// if all axes are finsihed, we're done
IF xFin AND yFin AND zFin THEN
	// reset local counters
	cX := 0;
	cY := 0;
	cZ := 0;
	fin := TRUE;
	RETURN;
END_IF

END_FUNCTION_BLOCK

// Device/Application/VG/FBs/VG_MOVE_TO_POS
(*
	Moves VG to certain position
	
Copyright (c) 2019 Manuel Goester, Michael Witt, Klaus Kammerer
Institute of Databases and Information Systems, Ulm University, Germany

Permission is hereby granted, free of charge, to any person obtaining a copy 
of this software and associated documentation files (the "Software"), to deal 
in the Software without restriction, including without limitation the rights 
to use, copy, modify, merge, publish, distribute, sublicense, and/or sell 
copies of the Software, and to permit persons to whom the Software is 
furnished to do so, subject to the following conditions:

The above copyright notice and this permission notice shall be included in 
all copies or substantial portions of the Software.

THE SOFTWARE IS PROVIDED "AS IS", WITHOUT WARRANTY OF ANY KIND, EXPRESS OR 
IMPLIED, INCLUDING BUT NOT LIMITED TO THE WARRANTIES OF MERCHANTABILITY, 
FITNESS FOR A PARTICULAR PURPOSE AND NONINFRINGEMENT. IN NO EVENT SHALL THE 
AUTHORS OR COPYRIGHT HOLDERS BE LIABLE FOR ANY CLAIM, DAMAGES OR OTHER 
LIABILITY, WHETHER IN AN ACTION OF CONTRACT, TORT OR OTHERWISE, ARISING FROM, 
OUT OF OR IN CONNECTION WITH THE SOFTWARE OR THE USE OR OTHER DEALINGS 
IN THE SOFTWARE.
*)
FUNCTION_BLOCK VG_MOVE_TO_POS
VAR_INPUT
	x: INT;
	y: INT;
	z: INT;
END_VAR
VAR_OUTPUT
END_VAR
VAR
	// finish flags
	xFin: BOOL := FALSE;
	yFin: BOOL := FALSE;
	zFin: BOOL := FALSE;
	fin: BOOL := FALSE;
	// true, if an impulse coming from the motor has been already counted
	xAlreadyCounted: BOOL := FALSE;
	yAlreadyCounted: BOOL := FALSE;
	zAlreadyCounted: BOOL := FALSE;
END_VAR

fin := FALSE;
// to handle negative counter values
IF VG.cX < 0 THEN
	VG.cX := 0;
END_IF
IF VG.cY < 0 THEN
	VG.cY := 0;
END_IF
IF VG.cZ < 0 THEN
	VG.cZ := 0;
END_IF

// X AXIS (Forward/Backward)
IF VG.cX = x THEN
	// if counter reached demanded position, we're done
	VG.mHorizontalForward := FALSE;
	VG.mHorizontalBackward := FALSE;
	xFin := TRUE;
ELSE
	xFin := FALSE;
	IF VG.cX < x AND NOT(xFin) THEN
		VG.mHorizontalForward := TRUE;
		VG.mHorizontalBackward := FALSE;
		IF VG.encHorizontal AND NOT(xAlreadyCounted) THEN
			VG.cX := VG.cX + 1;
			xAlreadyCounted := TRUE;
		ELSIF NOT(VG.encHorizontal) THEN
			xAlreadyCounted := FALSE;
		END_IF
	ELSIF VG.cX > x AND NOT(xFin) THEN
		VG.mHorizontalForward := FALSE;
		VG.mHorizontalBackward := TRUE;
		IF VG.encHorizontal AND NOT(xAlreadyCounted) THEN
			VG.cX := VG.cX - 1;
			xAlreadyCounted := TRUE;
		ELSIF NOT(VG.encHorizontal) THEN
			xAlreadyCounted := FALSE;
		END_IF
	END_IF
END_IF

// Y AXIS (Up/Down)
IF VG.cY = y THEN
	// if counter reached demanded position, we're done
	VG.mVerticalUp := FALSE;
	VG.mVerticalDown := FALSE;
	yFin := TRUE;
ELSE
	yFin := FALSE;
	IF VG.cY < y AND NOT(yFin) THEN
		VG.mVerticalDown := TRUE;
		VG.mVerticalUp := FALSE;
		IF VG.encVertical AND NOT(yAlreadyCounted) THEN
			VG.cY := VG.cY + 1;
			yAlreadyCounted := TRUE;
		ELSIF NOT(VG.encVertical) THEN
			yAlreadyCounted := FALSE;
		END_IF
	ELSIF VG.cY > y AND NOT(yFin) THEN
		VG.mVerticalUp := TRUE;
		VG.mVerticalDown := FALSE;
		IF VG.encVertical AND NOT(yAlreadyCounted) THEN
			VG.cY := VG.cY - 1;
			yAlreadyCounted := TRUE;
		ELSIF NOT(VG.encVertical) THEN
			yAlreadyCounted := FALSE;
		END_IF
	END_IF
END_IF

// Z AXIS (Rotation)
IF VG.cZ = z THEN
	// if counter reached demanded position, we're done
	VG.mRotationCClockwise := FALSE;
	VG.mRotationClockwise := FALSE;
	zFin := TRUE;
ELSE
	zFin := FALSE;
	IF VG.cZ < z AND NOT(zFin) THEN
		VG.mRotationCClockwise := TRUE;
		VG.mRotationClockwise := FALSE;
		IF VG.encRotation AND NOT(zAlreadyCounted) THEN
			VG.cZ := VG.cZ + 1;
			zAlreadyCounted := TRUE;
		ELSIF NOT(VG.encRotation) THEN
			zAlreadyCounted := FALSE;
		END_IF
	ELSIF VG.cZ > z AND NOT(zFin) THEN
		VG.mRotationCClockwise := FALSE;
		VG.mRotationClockwise := TRUE;
		IF VG.encRotation AND NOT(zAlreadyCounted) THEN
			VG.cZ := VG.cZ - 1;
			zAlreadyCounted := TRUE;
		ELSIF NOT(VG.encRotation) THEN
			zAlreadyCounted := FALSE;
		END_IF
	END_IF
END_IF

// if x and y axis are finsihed, we're done
IF xFin AND yFin AND zFin THEN
	fin := TRUE;
	RETURN;
END_IF

END_FUNCTION_BLOCK

// Device/Application/VG/VG_MULTI_MODE
PROGRAM VG_MULTI_MODE
VAR
	fin: BOOL;
	step: INT := 1;
	timer: TON;
	sorting_line_pos: INT := -1;
	vg_move_to_pos: VG_MOVE_TO_POS;
	vg_move: VG_MOVE;
END_VAR

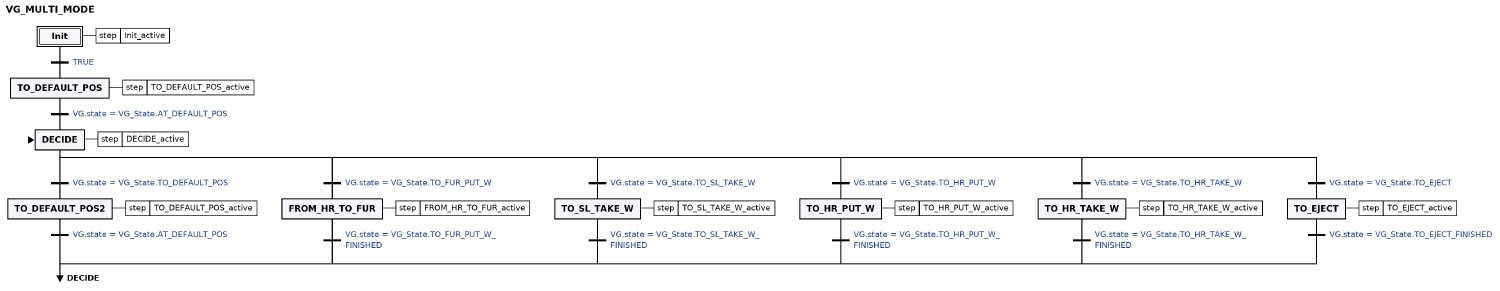
INITIAL_STEP Init:
    Init_active(N);  // step action
END_STEP
TRANSITION FROM Init TO TO_DEFAULT_POS
    := TRUE;
END_TRANSITION
STEP TO_DEFAULT_POS:
    TO_DEFAULT_POS_active(N);  // step action
END_STEP
TRANSITION FROM TO_DEFAULT_POS TO DECIDE
    := VG.state = VG_State.AT_DEFAULT_POS;
END_TRANSITION
STEP DECIDE:
    DECIDE_active(N);  // step action
END_STEP
TRANSITION FROM DECIDE TO TO_DEFAULT_POS2
    := VG.state = VG_State.TO_DEFAULT_POS;
END_TRANSITION
STEP TO_DEFAULT_POS2:
    TO_DEFAULT_POS_active(N);  // step action
END_STEP
TRANSITION FROM TO_DEFAULT_POS2 TO DECIDE
    := VG.state = VG_State.AT_DEFAULT_POS;
END_TRANSITION
TRANSITION FROM DECIDE TO FROM_HR_TO_FUR
    := VG.state = VG_State.TO_FUR_PUT_W;
END_TRANSITION
STEP FROM_HR_TO_FUR:
    FROM_HR_TO_FUR_active(N);  // step action
END_STEP
TRANSITION FROM FROM_HR_TO_FUR TO DECIDE
    := VG.state = VG_State.TO_FUR_PUT_W_FINISHED;
END_TRANSITION
TRANSITION FROM DECIDE TO TO_SL_TAKE_W
    := VG.state = VG_State.TO_SL_TAKE_W;
END_TRANSITION
STEP TO_SL_TAKE_W:
    TO_SL_TAKE_W_active(N);  // step action
END_STEP
TRANSITION FROM TO_SL_TAKE_W TO DECIDE
    := VG.state = VG_State.TO_SL_TAKE_W_FINISHED;
END_TRANSITION
TRANSITION FROM DECIDE TO TO_HR_PUT_W
    := VG.state = VG_State.TO_HR_PUT_W;
END_TRANSITION
STEP TO_HR_PUT_W:
    TO_HR_PUT_W_active(N);  // step action
END_STEP
TRANSITION FROM TO_HR_PUT_W TO DECIDE
    := VG.state = VG_State.TO_HR_PUT_W_FINISHED;
END_TRANSITION
TRANSITION FROM DECIDE TO TO_HR_TAKE_W
    := VG.state = VG_State.TO_HR_TAKE_W;
END_TRANSITION
STEP TO_HR_TAKE_W:
    TO_HR_TAKE_W_active(N);  // step action
END_STEP
TRANSITION FROM TO_HR_TAKE_W TO DECIDE
    := VG.state = VG_State.TO_HR_TAKE_W_FINISHED;
END_TRANSITION
TRANSITION FROM DECIDE TO TO_EJECT
    := VG.state = VG_State.TO_EJECT;
END_TRANSITION
STEP TO_EJECT:
    TO_EJECT_active(N);  // step action
END_STEP
TRANSITION FROM TO_EJECT TO DECIDE
    := VG.state = VG_State.TO_EJECT_FINISHED;
END_TRANSITION

ACTION TO_DEFAULT_POS_active:
(*
Copyright (c) 2019 Manuel Goester, Michael Witt, Klaus Kammerer
Institute of Databases and Information Systems, Ulm University, Germany

Permission is hereby granted, free of charge, to any person obtaining a copy 
of this software and associated documentation files (the "Software"), to deal 
in the Software without restriction, including without limitation the rights 
to use, copy, modify, merge, publish, distribute, sublicense, and/or sell 
copies of the Software, and to permit persons to whom the Software is 
furnished to do so, subject to the following conditions:

The above copyright notice and this permission notice shall be included in 
all copies or substantial portions of the Software.

THE SOFTWARE IS PROVIDED "AS IS", WITHOUT WARRANTY OF ANY KIND, EXPRESS OR 
IMPLIED, INCLUDING BUT NOT LIMITED TO THE WARRANTIES OF MERCHANTABILITY, 
FITNESS FOR A PARTICULAR PURPOSE AND NONINFRINGEMENT. IN NO EVENT SHALL THE 
AUTHORS OR COPYRIGHT HOLDERS BE LIABLE FOR ANY CLAIM, DAMAGES OR OTHER 
LIABILITY, WHETHER IN AN ACTION OF CONTRACT, TORT OR OTHERWISE, ARISING FROM, 
OUT OF OR IN CONNECTION WITH THE SOFTWARE OR THE USE OR OTHER DEALINGS 
IN THE SOFTWARE.
*)
// Brings VG to its default pos where sVertical = sHorizontal = sRotation = TRUE
// 1. y-Axis 2. z-Axis 3. rotation
IF NOT(VG.sVertical) THEN
	VG.mVerticalUp := TRUE;
ELSE
	VG.mVerticalUp := FALSE;
	// reset position counter
	VG.cY := 0;
	IF NOT(VG.sHorizontal) THEN
		VG.mHorizontalBackward := TRUE;
	ELSE
		VG.mHorizontalBackward := FALSE;
		// reset position counter
		VG.cX := 0;
		IF NOT(VG.sRotation) THEN
			VG.mRotationClockwise := TRUE;
		ELSE
			VG.mRotationClockwise := FALSE;
			// reset position counter
			VG.cZ := 0;
			
			// wait for 0.5 sec
			timer(IN:= TRUE, PT := T#0.5S);
			IF NOT(timer.Q = FALSE AND timer.IN) THEN
				timer(IN:=FALSE);
				
				// default pos reached
				VG.state := VG_State.AT_DEFAULT_POS;
			END_IF
		END_IF
	END_IF
END_IF
END_ACTION

ACTION DECIDE_active:
(*
Copyright (c) 2019 Manuel Goester, Michael Witt, Klaus Kammerer
Institute of Databases and Information Systems, Ulm University, Germany

Permission is hereby granted, free of charge, to any person obtaining a copy 
of this software and associated documentation files (the "Software"), to deal 
in the Software without restriction, including without limitation the rights 
to use, copy, modify, merge, publish, distribute, sublicense, and/or sell 
copies of the Software, and to permit persons to whom the Software is 
furnished to do so, subject to the following conditions:

The above copyright notice and this permission notice shall be included in 
all copies or substantial portions of the Software.

THE SOFTWARE IS PROVIDED "AS IS", WITHOUT WARRANTY OF ANY KIND, EXPRESS OR 
IMPLIED, INCLUDING BUT NOT LIMITED TO THE WARRANTIES OF MERCHANTABILITY, 
FITNESS FOR A PARTICULAR PURPOSE AND NONINFRINGEMENT. IN NO EVENT SHALL THE 
AUTHORS OR COPYRIGHT HOLDERS BE LIABLE FOR ANY CLAIM, DAMAGES OR OTHER 
LIABILITY, WHETHER IN AN ACTION OF CONTRACT, TORT OR OTHERWISE, ARISING FROM, 
OUT OF OR IN CONNECTION WITH THE SOFTWARE OR THE USE OR OTHER DEALINGS 
IN THE SOFTWARE.
*)
IF VG.state = VG_State.AT_HR THEN
	// this can happen if the batch job before was a single mode batch job. Then VG is already AT HR and is not in ready state
	VG.state := VG_State.TO_HR_TAKE_W;
ELSIF VG.state = VG_State.READY AND (HR.state = HR_State.GET_W AND HR.currW.state <> W_State.NULL) THEN
	// go to HR and take w
	VG.state := VG_State.TO_HR_TAKE_W;
ELSIF VG.state = VG_State.READY AND (NOT(SL.lbWhite) OR NOT(SL.lbRed) OR NOT(SL.lbBlue)) AND SL.currW.state <> W_State.NULL AND (NOT(HR.decidedToTakeANewW) OR HR.currW.state = W_State.NULL) THEN
	// go to SL and take w
	// bend VG pointers to workpiece being picked up
	VG.bIdx := SL.bIdx;
	VG.wIdx := SL.wIdx;
	VG.currW := TC.batchJobQueue.batchJobs[VG.bIdx].workpieces[VG.wIdx];
	VG.state := VG_State.TO_SL_TAKE_W;
ELSIF VG.state = VG_State.TO_SL_TAKE_W_FINISHED THEN
	// reset SL pointers
	SL.bIdx := 0;
	SL.wIdx := 0;
	SL.currW := TC.nullW;
	// at SL, w taken, decide if going to EJECT or HR
	IF VG.currW.format.ejectEnabled THEN
		// go to eject point and eject w
		VG.state := VG_State.TO_EJECT;
	ELSE
		// go to HR and put down w
		VG.state := VG_State.TO_HR_PUT_W;
	END_IF
ELSIF VG.state = VG_State.TO_HR_TAKE_W_FINISHED THEN
	// at HR, w taken, decide if going to FUR or EJECT
	IF VG.currW.format.ejectEnabled AND NOT(VG.currW.format.colorCheckEnabled OR VG.currW.format.furEnabled OR VG.currW.format.sawEnabled) THEN
		// go to eject point and eject w
		VG.state := VG_State.TO_EJECT;
	ELSE
		// go to FUR and put down w
		// but only if FUR-succer is at its default pos
		IF FUR.sSuckerPosRa THEN
			VG.state := VG_State.TO_FUR_PUT_W;
		END_IF
	END_IF
ELSIF VG.state = VG_State.TO_EJECT_FINISHED OR VG.state = VG_State.TO_FUR_PUT_W_FINISHED OR  VG.state = VG_State.TO_HR_PUT_W_FINISHED THEN
	// eject or putting w to FUR finished, back to default position for calibrating axes
	// likewise if VG put down w at HR
	VG.state := VG_State.TO_DEFAULT_POS;
ELSIF VG.state = VG_State.AT_DEFAULT_POS THEN
	// state = ready if VG is at default pos or if VG put down a w at HR --> VG is ready for next w
	VG.state := VG_state.READY;
	// reset own pointers
	VG.bIdx := 0;
	VG.wIdx := 0;
	VG.currW := TC.nullW;
END_IF
END_ACTION

ACTION FROM_HR_TO_FUR_active:
(*
Copyright (c) 2019 Manuel Goester, Michael Witt, Klaus Kammerer
Institute of Databases and Information Systems, Ulm University, Germany

Permission is hereby granted, free of charge, to any person obtaining a copy 
of this software and associated documentation files (the "Software"), to deal 
in the Software without restriction, including without limitation the rights 
to use, copy, modify, merge, publish, distribute, sublicense, and/or sell 
copies of the Software, and to permit persons to whom the Software is 
furnished to do so, subject to the following conditions:

The above copyright notice and this permission notice shall be included in 
all copies or substantial portions of the Software.

THE SOFTWARE IS PROVIDED "AS IS", WITHOUT WARRANTY OF ANY KIND, EXPRESS OR 
IMPLIED, INCLUDING BUT NOT LIMITED TO THE WARRANTIES OF MERCHANTABILITY, 
FITNESS FOR A PARTICULAR PURPOSE AND NONINFRINGEMENT. IN NO EVENT SHALL THE 
AUTHORS OR COPYRIGHT HOLDERS BE LIABLE FOR ANY CLAIM, DAMAGES OR OTHER 
LIABILITY, WHETHER IN AN ACTION OF CONTRACT, TORT OR OTHERWISE, ARISING FROM, 
OUT OF OR IN CONNECTION WITH THE SOFTWARE OR THE USE OR OTHER DEALINGS 
IN THE SOFTWARE.
*)
CASE step OF
	1:
		// x and z axis: move to FUR
		IF NOT(fin) THEN
			vg_move_to_pos(x := 131, y := 0, z := 137);
			fin := vg_move_to_pos.fin;
		ELSE
			fin := FALSE;
			step := step + 1;
		END_IF
	2:
		// y axis: move to FUR
		IF NOT(fin) THEN
			vg_move_to_pos(x := 131, y := 85, z := 137);
			fin := vg_move_to_pos.fin;
		ELSE
			fin := FALSE;
			step := step + 1;
		END_IF
	3:
		// open ventil to put down w onto waggon
		VG.valve := FALSE;
		step := step + 1;
	4:
		// wait 1 second to get sure w is not succed anymore
		timer(IN:= TRUE, PT:= T#1S);
		IF NOT(timer.Q = FALSE AND timer.IN) THEN
			// reset timer
			timer(IN:= FALSE);
			step := step + 1;
		END_IF
	5:
		// y axis: go up as far as possible
		IF NOT(VG.sVertical) THEN
			VG.mVerticalUp := TRUE;
		ELSE
			VG.mVerticalUp := FALSE;
			// reset y axis counter
			VG.cY := 0;
			// reset step counter
			step := 1;
			// bend FUR-Burner pointers to current workpiece of VG
			FUR.bIdxBurner := VG.bIdx;
			FUR.wIdxBurner := VG.wIdx;
			FUR.currWBurner := TC.batchJobQueue.batchJobs[FUR.bIdxBurner].workpieces[FUR.wIdxBurner];
			// finished
			VG.state := VG_State.TO_FUR_PUT_W_FINISHED;
		END_IF
	6:
	
END_CASE
END_ACTION

ACTION TO_SL_TAKE_W_active:
(*
Copyright (c) 2019 Manuel Goester, Michael Witt, Klaus Kammerer
Institute of Databases and Information Systems, Ulm University, Germany

Permission is hereby granted, free of charge, to any person obtaining a copy 
of this software and associated documentation files (the "Software"), to deal 
in the Software without restriction, including without limitation the rights 
to use, copy, modify, merge, publish, distribute, sublicense, and/or sell 
copies of the Software, and to permit persons to whom the Software is 
furnished to do so, subject to the following conditions:

The above copyright notice and this permission notice shall be included in 
all copies or substantial portions of the Software.

THE SOFTWARE IS PROVIDED "AS IS", WITHOUT WARRANTY OF ANY KIND, EXPRESS OR 
IMPLIED, INCLUDING BUT NOT LIMITED TO THE WARRANTIES OF MERCHANTABILITY, 
FITNESS FOR A PARTICULAR PURPOSE AND NONINFRINGEMENT. IN NO EVENT SHALL THE 
AUTHORS OR COPYRIGHT HOLDERS BE LIABLE FOR ANY CLAIM, DAMAGES OR OTHER 
LIABILITY, WHETHER IN AN ACTION OF CONTRACT, TORT OR OTHERWISE, ARISING FROM, 
OUT OF OR IN CONNECTION WITH THE SOFTWARE OR THE USE OR OTHER DEALINGS 
IN THE SOFTWARE.
*)
CASE step OF
	1:
		IF NOT(SL.currW.format.ejectEnabled) THEN
			// set flag to inform HR that VG is taking a w to bring it back to HR
			VG.storeW := TRUE;
			//VG.bIdx := SL.bIdx;
			//VG.wIdx := SL.wIdx;
			//VG.currW := TC.batchJobQueue.batchJobs[VG.bIdx].workpieces[VG.wIdx];
		END_IF
		// select sorting line pos
		IF 	TC.batchJobQueue.batchJobs[SL.bIdx].workpieces[SL.wIdx].format.colorCheckEnabled THEN
			IF TC.batchJobQueue.batchJobs[SL.bIdx].workpieces[SL.wIdx].color = 'white' AND NOT(SL.lbWhite) THEN
				sorting_line_pos := 1;
			ELSIF TC.batchJobQueue.batchJobs[SL.bIdx].workpieces[SL.wIdx].color = 'red' AND NOT(SL.lbRed) THEN
				sorting_line_pos := 2;
			ELSIF TC.batchJobQueue.batchJobs[SL.bIdx].workpieces[SL.wIdx].color = 'blue' AND NOT(SL.lbBlue) THEN
				sorting_line_pos := 3;
			END_IF
		ELSE
			// when color was not checked
			sorting_line_pos := 1;
		END_IF
		step := step + 1;
	2:
		// x and z axis: move to SL
		IF NOT(fin) THEN
			CASE sorting_line_pos OF
				1:
					vg_move_to_pos(x := 58, y := 0, z := 69);
				2:
					vg_move_to_pos(x := 63, y := 0, z := 57);
				3:
					vg_move_to_pos(x := 87, y := 0, z := 47);
			END_CASE
		fin := vg_move_to_pos.fin;
		ELSE
			fin := FALSE;
			step := step + 1;
		END_IF
	3:
		// y axis: move to SL
		IF NOT(fin) THEN
			CASE sorting_line_pos OF
				1:
					vg_move_to_pos(x := 58, y := 125, z := 69);
				2:
					vg_move_to_pos(x := 63, y := 125, z := 57);
				3:
					vg_move_to_pos(x := 87, y := 125, z := 47);
			END_CASE
		fin := vg_move_to_pos.fin;
		ELSE
			fin := FALSE;
			step := step + 1;
		END_IF
	4:
		// succ workpiece at SL
		VG.valve := TRUE;
		timer(IN:= TRUE, PT:= T#2S);
		IF timer.Q = FALSE AND timer.IN THEN
			// go
			VG.compressor := TRUE;
		ELSE
			// stop
			VG.compressor := FALSE;
			// reset timer
			timer(IN:= FALSE);
			step := step + 1;
		END_IF
	5:
		// y axis: go up as far as possible
		IF NOT(VG.sVertical) THEN
			VG.mVerticalUp := TRUE;
		ELSE
			VG.mVerticalUp := FALSE;
			// reset y axis counter
			VG.cY := 0;
			// reset step counter
			step := 1;
			// reset sorting line pos
			sorting_line_pos := -1;
			// finished
			VG.state := VG_State.TO_SL_TAKE_W_FINISHED;
		END_IF
END_CASE
END_ACTION

ACTION TO_HR_PUT_W_active:
(*
Copyright (c) 2019 Manuel Goester, Michael Witt, Klaus Kammerer
Institute of Databases and Information Systems, Ulm University, Germany

Permission is hereby granted, free of charge, to any person obtaining a copy 
of this software and associated documentation files (the "Software"), to deal 
in the Software without restriction, including without limitation the rights 
to use, copy, modify, merge, publish, distribute, sublicense, and/or sell 
copies of the Software, and to permit persons to whom the Software is 
furnished to do so, subject to the following conditions:

The above copyright notice and this permission notice shall be included in 
all copies or substantial portions of the Software.

THE SOFTWARE IS PROVIDED "AS IS", WITHOUT WARRANTY OF ANY KIND, EXPRESS OR 
IMPLIED, INCLUDING BUT NOT LIMITED TO THE WARRANTIES OF MERCHANTABILITY, 
FITNESS FOR A PARTICULAR PURPOSE AND NONINFRINGEMENT. IN NO EVENT SHALL THE 
AUTHORS OR COPYRIGHT HOLDERS BE LIABLE FOR ANY CLAIM, DAMAGES OR OTHER 
LIABILITY, WHETHER IN AN ACTION OF CONTRACT, TORT OR OTHERWISE, ARISING FROM, 
OUT OF OR IN CONNECTION WITH THE SOFTWARE OR THE USE OR OTHER DEALINGS 
IN THE SOFTWARE.
*)
CASE step OF
	1:
		// x and z axis: move to HR
		IF NOT(fin) THEN
			vg_move_to_pos(x := 27, y := 0, z := 206);
			fin := vg_move_to_pos.fin;
		ELSE
			fin := FALSE;
			step := step + 1;
		END_IF
	2:
		// box without workpiece arrived, wait 0.5 sec to be sure
		IF NOT(HR.lbOut) AND HR.state = HR_State.WAIT_FOR_VG_TO_BRING_W THEN
			timer(IN:= TRUE, PT:= T#0.5S);
			IF NOT(timer.Q = FALSE AND timer.IN) THEN
				timer(IN:= FALSE);
				step := step + 1;
			END_IF
		END_IF
	3:
		// y axis: move down at HR
		IF NOT(fin) THEN
			vg_move_to_pos(x:=27, y:=40, z:=206);
			fin := vg_move_to_pos.fin;
		ELSE
			fin := FALSE;
			step := step + 1;
		END_IF
	4:
		// open ventil
		VG.valve := FALSE;
		step := step + 1;
	5:
		timer(IN:= TRUE, PT:= T#1S);
		IF NOT(timer.Q = FALSE AND timer.IN) THEN
			// reset timer
			timer(IN:= FALSE);
			// go to next step
			step := step + 1;
		END_IF
	6:
		// y axis: go up as far as possible
		IF NOT(VG.sVertical) THEN
			VG.mVerticalUp := TRUE;
		ELSE
			VG.mVerticalUp := FALSE;
			// reset y axis counter
			VG.cY := 0;
			// reset step counter
			step := 1;
			// finished
			VG.state := VG_State.TO_HR_PUT_W_FINISHED;
		END_IF
END_CASE
END_ACTION

ACTION TO_HR_TAKE_W_active:
(*
Copyright (c) 2019 Manuel Goester, Michael Witt, Klaus Kammerer
Institute of Databases and Information Systems, Ulm University, Germany

Permission is hereby granted, free of charge, to any person obtaining a copy 
of this software and associated documentation files (the "Software"), to deal 
in the Software without restriction, including without limitation the rights 
to use, copy, modify, merge, publish, distribute, sublicense, and/or sell 
copies of the Software, and to permit persons to whom the Software is 
furnished to do so, subject to the following conditions:

The above copyright notice and this permission notice shall be included in 
all copies or substantial portions of the Software.

THE SOFTWARE IS PROVIDED "AS IS", WITHOUT WARRANTY OF ANY KIND, EXPRESS OR 
IMPLIED, INCLUDING BUT NOT LIMITED TO THE WARRANTIES OF MERCHANTABILITY, 
FITNESS FOR A PARTICULAR PURPOSE AND NONINFRINGEMENT. IN NO EVENT SHALL THE 
AUTHORS OR COPYRIGHT HOLDERS BE LIABLE FOR ANY CLAIM, DAMAGES OR OTHER 
LIABILITY, WHETHER IN AN ACTION OF CONTRACT, TORT OR OTHERWISE, ARISING FROM, 
OUT OF OR IN CONNECTION WITH THE SOFTWARE OR THE USE OR OTHER DEALINGS 
IN THE SOFTWARE.
*)
CASE step OF
	1:
		// x and z axis: move to HR
		IF NOT(fin) THEN
			vg_move_to_pos(x := 27, y := 0, z := 206);
			fin := vg_move_to_pos.fin;
		ELSE
			fin := FALSE;
			step := step + 1;
		END_IF
	2:
		IF NOT(HR.lbOut) THEN
			// box with workpiece arrived, wait 0.5 sec to be sure
			timer(IN:= TRUE, PT:= T#0.5S);
			IF NOT(timer.Q = FALSE AND timer.IN) THEN
				timer(IN:= FALSE);
				step := step + 1;
			END_IF		
		END_IF
	3:
		// y axis: move down at HR
		IF NOT(fin) THEN
			vg_move_to_pos(x:=27, y:=40, z:=206);
			fin := vg_move_to_pos.fin;
		ELSE
			fin := FALSE;
			step := step + 1;
		END_IF
	4:
		// succ w at HR
		VG.valve := TRUE;
		timer(IN:= TRUE, PT:= T#2S);
		IF timer.Q = FALSE AND timer.IN THEN
			// go
			VG.compressor := TRUE;
		ELSE
			// stop
			VG.compressor := FALSE;
			// reset timer
			timer(IN:= FALSE);
			step := step + 1;
		END_IF	
	5:
		// y axis: go up as far as possible
		IF NOT(VG.sVertical) THEN
			VG.mVerticalUp := TRUE;
		ELSE
			VG.mVerticalUp := FALSE;
			// reset y axis counter
			VG.cY := 0;
			// reset step counter
			step := 1;
			// finished
			VG.state := VG_State.TO_HR_TAKE_W_FINISHED;
		END_IF
END_CASE
END_ACTION

ACTION TO_EJECT_active:
(*
Copyright (c) 2019 Manuel Goester, Michael Witt, Klaus Kammerer
Institute of Databases and Information Systems, Ulm University, Germany

Permission is hereby granted, free of charge, to any person obtaining a copy 
of this software and associated documentation files (the "Software"), to deal 
in the Software without restriction, including without limitation the rights 
to use, copy, modify, merge, publish, distribute, sublicense, and/or sell 
copies of the Software, and to permit persons to whom the Software is 
furnished to do so, subject to the following conditions:

The above copyright notice and this permission notice shall be included in 
all copies or substantial portions of the Software.

THE SOFTWARE IS PROVIDED "AS IS", WITHOUT WARRANTY OF ANY KIND, EXPRESS OR 
IMPLIED, INCLUDING BUT NOT LIMITED TO THE WARRANTIES OF MERCHANTABILITY, 
FITNESS FOR A PARTICULAR PURPOSE AND NONINFRINGEMENT. IN NO EVENT SHALL THE 
AUTHORS OR COPYRIGHT HOLDERS BE LIABLE FOR ANY CLAIM, DAMAGES OR OTHER 
LIABILITY, WHETHER IN AN ACTION OF CONTRACT, TORT OR OTHERWISE, ARISING FROM, 
OUT OF OR IN CONNECTION WITH THE SOFTWARE OR THE USE OR OTHER DEALINGS 
IN THE SOFTWARE.
*)
CASE step OF
	1:
		// x and z axis: move to EJECT
		IF NOT(fin) THEN
			IF VG.currW.color = 'white' THEN
				// go to eject point 1
				vg_move_to_pos(x := 25, y := 0, z := 2);
			ELSIF VG.currW.color = 'red' THEN
				// go to eject point 2
				vg_move_to_pos(x := 30, y := 0, z := 15);
			ELSIF VG.currW.color = 'blue' THEN
				// go to eject point 3
				vg_move_to_pos(x := 49, y := 0, z := 23);
			ELSE
				// if color 'unknown' then eject to white eject point
				// go to eject point 1
				vg_move_to_pos(x := 25, y := 0, z := 2);
			END_IF
			fin := vg_move_to_pos.fin;
		ELSE
			fin := FALSE;
			step := step + 1;
		END_IF
	2:
		// x and z axis: move to EJECT
		IF NOT(fin) THEN
			IF VG.currW.color = 'white' THEN
				// go to eject point 1
				vg_move_to_pos(x := 25, y := 133, z := 2);
			ELSIF VG.currW.color = 'red' THEN
				// go to eject point 2
				vg_move_to_pos(x := 30, y := 133, z := 15);
			ELSIF VG.currW.color = 'blue' THEN
				// go to eject point 3
				vg_move_to_pos(x := 49, y := 133, z := 23);
			ELSE
				// if color 'unknown' then eject to white eject point
				// go to eject point 1
				vg_move_to_pos(x := 25, y := 133, z := 2);
			END_IF
			fin := vg_move_to_pos.fin;
		ELSE
			fin := FALSE;
			step := step + 1;
		END_IF
	3:
		// open valve to drop w
		VG.valve := FALSE;
		timer(IN:= TRUE, PT:= T#1S);
		IF NOT(timer.Q = FALSE AND timer.IN) THEN
			// reset timer
			timer(IN:= FALSE);
			// reset step counter
			step := 1;
			// finished
			VG.state := VG_State.TO_EJECT_FINISHED;
		END_IF
END_CASE
END_ACTION

ACTION Init_active:
(*
Copyright (c) 2019 Manuel Goester, Michael Witt, Klaus Kammerer
Institute of Databases and Information Systems, Ulm University, Germany

Permission is hereby granted, free of charge, to any person obtaining a copy 
of this software and associated documentation files (the "Software"), to deal 
in the Software without restriction, including without limitation the rights 
to use, copy, modify, merge, publish, distribute, sublicense, and/or sell 
copies of the Software, and to permit persons to whom the Software is 
furnished to do so, subject to the following conditions:

The above copyright notice and this permission notice shall be included in 
all copies or substantial portions of the Software.

THE SOFTWARE IS PROVIDED "AS IS", WITHOUT WARRANTY OF ANY KIND, EXPRESS OR 
IMPLIED, INCLUDING BUT NOT LIMITED TO THE WARRANTIES OF MERCHANTABILITY, 
FITNESS FOR A PARTICULAR PURPOSE AND NONINFRINGEMENT. IN NO EVENT SHALL THE 
AUTHORS OR COPYRIGHT HOLDERS BE LIABLE FOR ANY CLAIM, DAMAGES OR OTHER 
LIABILITY, WHETHER IN AN ACTION OF CONTRACT, TORT OR OTHERWISE, ARISING FROM, 
OUT OF OR IN CONNECTION WITH THE SOFTWARE OR THE USE OR OTHER DEALINGS 
IN THE SOFTWARE.
*)
step := 1;
END_ACTION

END_PROGRAM

// Device/Application/SL/SL_SINGLE_MODE
PROGRAM SL_SINGLE_MODE
VAR
	sl_fb: SL_FB;
	step: INT := 1;
	fin: BOOL;
END_VAR

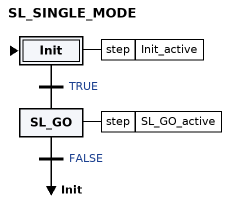
INITIAL_STEP Init:
    Init_active(N);  // step action
END_STEP
TRANSITION FROM Init TO SL_GO
    := TRUE;
END_TRANSITION
STEP SL_GO:
    SL_GO_active(N);  // step action
END_STEP
TRANSITION FROM SL_GO TO Init
    := FALSE;
END_TRANSITION

ACTION Init_active:
(*
Copyright (c) 2019 Manuel Goester, Michael Witt, Klaus Kammerer
Institute of Databases and Information Systems, Ulm University, Germany

Permission is hereby granted, free of charge, to any person obtaining a copy 
of this software and associated documentation files (the "Software"), to deal 
in the Software without restriction, including without limitation the rights 
to use, copy, modify, merge, publish, distribute, sublicense, and/or sell 
copies of the Software, and to permit persons to whom the Software is 
furnished to do so, subject to the following conditions:

The above copyright notice and this permission notice shall be included in 
all copies or substantial portions of the Software.

THE SOFTWARE IS PROVIDED "AS IS", WITHOUT WARRANTY OF ANY KIND, EXPRESS OR 
IMPLIED, INCLUDING BUT NOT LIMITED TO THE WARRANTIES OF MERCHANTABILITY, 
FITNESS FOR A PARTICULAR PURPOSE AND NONINFRINGEMENT. IN NO EVENT SHALL THE 
AUTHORS OR COPYRIGHT HOLDERS BE LIABLE FOR ANY CLAIM, DAMAGES OR OTHER 
LIABILITY, WHETHER IN AN ACTION OF CONTRACT, TORT OR OTHERWISE, ARISING FROM, 
OUT OF OR IN CONNECTION WITH THE SOFTWARE OR THE USE OR OTHER DEALINGS 
IN THE SOFTWARE.
*)
SL.state := SL_State.WAITING_FOR_W;
END_ACTION

ACTION SL_GO_active:
(*
Copyright (c) 2019 Manuel Goester, Michael Witt, Klaus Kammerer
Institute of Databases and Information Systems, Ulm University, Germany

Permission is hereby granted, free of charge, to any person obtaining a copy 
of this software and associated documentation files (the "Software"), to deal 
in the Software without restriction, including without limitation the rights 
to use, copy, modify, merge, publish, distribute, sublicense, and/or sell 
copies of the Software, and to permit persons to whom the Software is 
furnished to do so, subject to the following conditions:

The above copyright notice and this permission notice shall be included in 
all copies or substantial portions of the Software.

THE SOFTWARE IS PROVIDED "AS IS", WITHOUT WARRANTY OF ANY KIND, EXPRESS OR 
IMPLIED, INCLUDING BUT NOT LIMITED TO THE WARRANTIES OF MERCHANTABILITY, 
FITNESS FOR A PARTICULAR PURPOSE AND NONINFRINGEMENT. IN NO EVENT SHALL THE 
AUTHORS OR COPYRIGHT HOLDERS BE LIABLE FOR ANY CLAIM, DAMAGES OR OTHER 
LIABILITY, WHETHER IN AN ACTION OF CONTRACT, TORT OR OTHERWISE, ARISING FROM, 
OUT OF OR IN CONNECTION WITH THE SOFTWARE OR THE USE OR OTHER DEALINGS 
IN THE SOFTWARE.
*)
CASE step OF
	1:
		IF SL.state = SL_State.W_RECEIVED THEN
			step := step + 1;
		END_IF
	2:
		IF NOT(fin) THEN
			sl_fb();
			fin := sl_fb.fin;
		ELSE
			// wait for VG to pick up w
			SL.state := SL_State.WAITING_FOR_VG_TO_PICK_UP_W;
			step := step + 1;
		END_IF
	3:
		// reset own pointers
		SL.bIdx := 0;
		SL.wIdx := 0;
		// reset fin
		fin := FALSE;
		step := 1;
		SL.state := SL_State.WAITING_FOR_W;
END_CASE
END_ACTION

END_PROGRAM

// Device/Application/SL/FBs/SL_FB
(*
	Implements the functionality of sorting line
*)
FUNCTION_BLOCK SL_FB
VAR_INPUT
END_VAR
VAR_OUTPUT
END_VAR
VAR
	trigger : INT;
	puls_temp : INT := 0;
	counter_puls : INT;
	white : BOOL;
	red : BOOL;
	blue : BOOL;
	
	color_value : DINT;
	
	rack_white : INT := 0;
	rack_red : INT := 0;
	rack_blue : INT := 0;
	
	timer : TON;
	passed: BOOL;
	fin: BOOL;
END_VAR

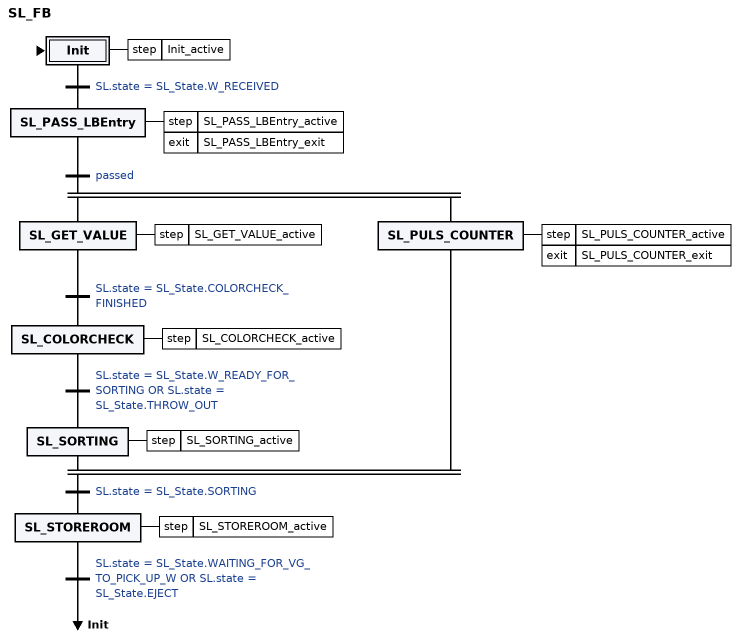
INITIAL_STEP Init:
    Init_active(N);  // step action
END_STEP
TRANSITION FROM Init TO SL_PASS_LBEntry
    := SL.state = SL_State.W_RECEIVED;
END_TRANSITION
STEP SL_PASS_LBEntry:
    SL_PASS_LBEntry_active(N);  // step action
    SL_PASS_LBEntry_exit(P0);  // exit action
END_STEP
TRANSITION FROM SL_PASS_LBEntry TO (SL_GET_VALUE, SL_PULS_COUNTER)
    := passed;
END_TRANSITION
STEP SL_GET_VALUE:
    SL_GET_VALUE_active(N);  // step action
END_STEP
TRANSITION FROM SL_GET_VALUE TO SL_COLORCHECK
    := SL.state = SL_State.COLORCHECK_FINISHED;
END_TRANSITION
STEP SL_COLORCHECK:
    SL_COLORCHECK_active(N);  // step action
END_STEP
TRANSITION FROM SL_COLORCHECK TO SL_SORTING
    := SL.state = SL_State.W_READY_FOR_SORTING OR SL.state = SL_State.THROW_OUT;
END_TRANSITION
STEP SL_SORTING:
    SL_SORTING_active(N);  // step action
END_STEP
STEP SL_PULS_COUNTER:
    SL_PULS_COUNTER_active(N);  // step action
    SL_PULS_COUNTER_exit(P0);  // exit action
END_STEP
TRANSITION FROM (SL_SORTING, SL_PULS_COUNTER) TO SL_STOREROOM
    := SL.state = SL_State.SORTING;
END_TRANSITION
STEP SL_STOREROOM:
    SL_STOREROOM_active(N);  // step action
END_STEP
TRANSITION FROM SL_STOREROOM TO Init
    := SL.state = SL_State.WAITING_FOR_VG_TO_PICK_UP_W OR SL.state = SL_State.EJECT;
END_TRANSITION

ACTION Init_active:
(*
Copyright (c) 2019 Manuel Goester, Michael Witt, Klaus Kammerer
Institute of Databases and Information Systems, Ulm University, Germany

Permission is hereby granted, free of charge, to any person obtaining a copy 
of this software and associated documentation files (the "Software"), to deal 
in the Software without restriction, including without limitation the rights 
to use, copy, modify, merge, publish, distribute, sublicense, and/or sell 
copies of the Software, and to permit persons to whom the Software is 
furnished to do so, subject to the following conditions:

The above copyright notice and this permission notice shall be included in 
all copies or substantial portions of the Software.

THE SOFTWARE IS PROVIDED "AS IS", WITHOUT WARRANTY OF ANY KIND, EXPRESS OR 
IMPLIED, INCLUDING BUT NOT LIMITED TO THE WARRANTIES OF MERCHANTABILITY, 
FITNESS FOR A PARTICULAR PURPOSE AND NONINFRINGEMENT. IN NO EVENT SHALL THE 
AUTHORS OR COPYRIGHT HOLDERS BE LIABLE FOR ANY CLAIM, DAMAGES OR OTHER 
LIABILITY, WHETHER IN AN ACTION OF CONTRACT, TORT OR OTHERWISE, ARISING FROM, 
OUT OF OR IN CONNECTION WITH THE SOFTWARE OR THE USE OR OTHER DEALINGS 
IN THE SOFTWARE.
*)
trigger := 0;
puls_temp := 0;
counter_puls := 0;
white := FALSE;
red := FALSE;
blue := FALSE;

color_value := 4000000;

timer(IN:=FALSE);
fin := FALSE;

SL.mConveyorBelt := TRUE;
END_ACTION

ACTION SL_COLORCHECK_active:
(*
Copyright (c) 2019 Manuel Goester, Michael Witt, Klaus Kammerer
Institute of Databases and Information Systems, Ulm University, Germany

Permission is hereby granted, free of charge, to any person obtaining a copy 
of this software and associated documentation files (the "Software"), to deal 
in the Software without restriction, including without limitation the rights 
to use, copy, modify, merge, publish, distribute, sublicense, and/or sell 
copies of the Software, and to permit persons to whom the Software is 
furnished to do so, subject to the following conditions:

The above copyright notice and this permission notice shall be included in 
all copies or substantial portions of the Software.

THE SOFTWARE IS PROVIDED "AS IS", WITHOUT WARRANTY OF ANY KIND, EXPRESS OR 
IMPLIED, INCLUDING BUT NOT LIMITED TO THE WARRANTIES OF MERCHANTABILITY, 
FITNESS FOR A PARTICULAR PURPOSE AND NONINFRINGEMENT. IN NO EVENT SHALL THE 
AUTHORS OR COPYRIGHT HOLDERS BE LIABLE FOR ANY CLAIM, DAMAGES OR OTHER 
LIABILITY, WHETHER IN AN ACTION OF CONTRACT, TORT OR OTHERWISE, ARISING FROM, 
OUT OF OR IN CONNECTION WITH THE SOFTWARE OR THE USE OR OTHER DEALINGS 
IN THE SOFTWARE.
*)
IF color_value > 2000000 AND color_value < 2558000 THEN//weis: 2630000
	TC.batchJobQueue.batchJobs[SL.bIdx].workpieces[SL.wIdx].color := 'white';
	white := TRUE;
	red := FALSE;
	blue := FALSE;
	SL.state := SL_State.W_READY_FOR_SORTING;
END_IF
IF color_value > 2558001 AND color_value < 3000000 THEN//rot: 2801000
	TC.batchJobQueue.batchJobs[SL.bIdx].workpieces[SL.wIdx].color := 'red';
	white := FALSE;
	red := TRUE;
	blue := FALSE;
	SL.state := SL_State.W_READY_FOR_SORTING;
END_IF
IF color_value > 3400000 AND color_value < 3600000 THEN//blau: 3546000
	TC.batchJobQueue.batchJobs[SL.bIdx].workpieces[SL.wIdx].color := 'blue';
	white := FALSE;
	red := FALSE;
	blue := TRUE;
	SL.state := SL_State.W_READY_FOR_SORTING;
END_IF
IF color_value > 3600000 OR color_value < 2000000 THEN//unknown
	TC.batchJobQueue.batchJobs[SL.bIdx].workpieces[SL.wIdx].color := 'unknown';
	white := FALSE;
	red := FALSE;
	blue := FALSE;
	SL.state := SL_State.THROW_OUT; 
END_IF

SL.mConveyorBelt := TRUE;
END_ACTION

ACTION SL_GET_VALUE_active:
(*
Copyright (c) 2019 Manuel Goester, Michael Witt, Klaus Kammerer
Institute of Databases and Information Systems, Ulm University, Germany

Permission is hereby granted, free of charge, to any person obtaining a copy 
of this software and associated documentation files (the "Software"), to deal 
in the Software without restriction, including without limitation the rights 
to use, copy, modify, merge, publish, distribute, sublicense, and/or sell 
copies of the Software, and to permit persons to whom the Software is 
furnished to do so, subject to the following conditions:

The above copyright notice and this permission notice shall be included in 
all copies or substantial portions of the Software.

THE SOFTWARE IS PROVIDED "AS IS", WITHOUT WARRANTY OF ANY KIND, EXPRESS OR 
IMPLIED, INCLUDING BUT NOT LIMITED TO THE WARRANTIES OF MERCHANTABILITY, 
FITNESS FOR A PARTICULAR PURPOSE AND NONINFRINGEMENT. IN NO EVENT SHALL THE 
AUTHORS OR COPYRIGHT HOLDERS BE LIABLE FOR ANY CLAIM, DAMAGES OR OTHER 
LIABILITY, WHETHER IN AN ACTION OF CONTRACT, TORT OR OTHERWISE, ARISING FROM, 
OUT OF OR IN CONNECTION WITH THE SOFTWARE OR THE USE OR OTHER DEALINGS 
IN THE SOFTWARE.
*)
IF NOT(SL.lbAfterColorSensor) THEN
	SL.state := SL_State.COLORCHECK_FINISHED;
ELSE
	SL.state := SL_State.W_AT_COLORCHECK;
	IF SL.colorSensor < color_value THEN
		color_value := SL.colorSensor;
	END_IF
END_IF 

SL.mConveyorBelt := TRUE;
END_ACTION

ACTION SL_PASS_LBEntry_active:
(*
Copyright (c) 2019 Manuel Goester, Michael Witt, Klaus Kammerer
Institute of Databases and Information Systems, Ulm University, Germany

Permission is hereby granted, free of charge, to any person obtaining a copy 
of this software and associated documentation files (the "Software"), to deal 
in the Software without restriction, including without limitation the rights 
to use, copy, modify, merge, publish, distribute, sublicense, and/or sell 
copies of the Software, and to permit persons to whom the Software is 
furnished to do so, subject to the following conditions:

The above copyright notice and this permission notice shall be included in 
all copies or substantial portions of the Software.

THE SOFTWARE IS PROVIDED "AS IS", WITHOUT WARRANTY OF ANY KIND, EXPRESS OR 
IMPLIED, INCLUDING BUT NOT LIMITED TO THE WARRANTIES OF MERCHANTABILITY, 
FITNESS FOR A PARTICULAR PURPOSE AND NONINFRINGEMENT. IN NO EVENT SHALL THE 
AUTHORS OR COPYRIGHT HOLDERS BE LIABLE FOR ANY CLAIM, DAMAGES OR OTHER 
LIABILITY, WHETHER IN AN ACTION OF CONTRACT, TORT OR OTHERWISE, ARISING FROM, 
OUT OF OR IN CONNECTION WITH THE SOFTWARE OR THE USE OR OTHER DEALINGS 
IN THE SOFTWARE.
*)
IF NOT(SL.lbEntry) AND trigger < 1 THEN
	trigger := trigger + 1;
	SL.state := SL_State.W_AT_LB;
END_IF

IF lbEntry AND trigger >= 1 THEN
	passed := TRUE;
END_IF

SL.mConveyorBelt := TRUE;
END_ACTION

ACTION SL_PASS_LBEntry_exit:
(*
Copyright (c) 2019 Manuel Goester, Michael Witt, Klaus Kammerer
Institute of Databases and Information Systems, Ulm University, Germany

Permission is hereby granted, free of charge, to any person obtaining a copy 
of this software and associated documentation files (the "Software"), to deal 
in the Software without restriction, including without limitation the rights 
to use, copy, modify, merge, publish, distribute, sublicense, and/or sell 
copies of the Software, and to permit persons to whom the Software is 
furnished to do so, subject to the following conditions:

The above copyright notice and this permission notice shall be included in 
all copies or substantial portions of the Software.

THE SOFTWARE IS PROVIDED "AS IS", WITHOUT WARRANTY OF ANY KIND, EXPRESS OR 
IMPLIED, INCLUDING BUT NOT LIMITED TO THE WARRANTIES OF MERCHANTABILITY, 
FITNESS FOR A PARTICULAR PURPOSE AND NONINFRINGEMENT. IN NO EVENT SHALL THE 
AUTHORS OR COPYRIGHT HOLDERS BE LIABLE FOR ANY CLAIM, DAMAGES OR OTHER 
LIABILITY, WHETHER IN AN ACTION OF CONTRACT, TORT OR OTHERWISE, ARISING FROM, 
OUT OF OR IN CONNECTION WITH THE SOFTWARE OR THE USE OR OTHER DEALINGS 
IN THE SOFTWARE.
*)
passed := FALSE;
puls_temp := 0;
counter_puls := 0;
END_ACTION

ACTION SL_PULS_COUNTER_active:
(*
Copyright (c) 2019 Manuel Goester, Michael Witt, Klaus Kammerer
Institute of Databases and Information Systems, Ulm University, Germany

Permission is hereby granted, free of charge, to any person obtaining a copy 
of this software and associated documentation files (the "Software"), to deal 
in the Software without restriction, including without limitation the rights 
to use, copy, modify, merge, publish, distribute, sublicense, and/or sell 
copies of the Software, and to permit persons to whom the Software is 
furnished to do so, subject to the following conditions:

The above copyright notice and this permission notice shall be included in 
all copies or substantial portions of the Software.

THE SOFTWARE IS PROVIDED "AS IS", WITHOUT WARRANTY OF ANY KIND, EXPRESS OR 
IMPLIED, INCLUDING BUT NOT LIMITED TO THE WARRANTIES OF MERCHANTABILITY, 
FITNESS FOR A PARTICULAR PURPOSE AND NONINFRINGEMENT. IN NO EVENT SHALL THE 
AUTHORS OR COPYRIGHT HOLDERS BE LIABLE FOR ANY CLAIM, DAMAGES OR OTHER 
LIABILITY, WHETHER IN AN ACTION OF CONTRACT, TORT OR OTHERWISE, ARISING FROM, 
OUT OF OR IN CONNECTION WITH THE SOFTWARE OR THE USE OR OTHER DEALINGS 
IN THE SOFTWARE.
*)
//count convoyorbelt buttons
IF SL.mConveyorBelt AND SL.iFeeler THEN //button push
	IF puls_temp = 0 THEN
		counter_puls := counter_puls +1;
	END_IF
	
	puls_temp := puls_temp +1;
END_IF

IF puls_temp > 0 AND SL.mConveyorBelt AND NOT(iFeeler) THEN // button release
	puls_temp := 0;
	counter_puls := counter_puls +1;
END_IF
END_ACTION

ACTION SL_PULS_COUNTER_exit:
(*
Copyright (c) 2019 Manuel Goester, Michael Witt, Klaus Kammerer
Institute of Databases and Information Systems, Ulm University, Germany

Permission is hereby granted, free of charge, to any person obtaining a copy 
of this software and associated documentation files (the "Software"), to deal 
in the Software without restriction, including without limitation the rights 
to use, copy, modify, merge, publish, distribute, sublicense, and/or sell 
copies of the Software, and to permit persons to whom the Software is 
furnished to do so, subject to the following conditions:

The above copyright notice and this permission notice shall be included in 
all copies or substantial portions of the Software.

THE SOFTWARE IS PROVIDED "AS IS", WITHOUT WARRANTY OF ANY KIND, EXPRESS OR 
IMPLIED, INCLUDING BUT NOT LIMITED TO THE WARRANTIES OF MERCHANTABILITY, 
FITNESS FOR A PARTICULAR PURPOSE AND NONINFRINGEMENT. IN NO EVENT SHALL THE 
AUTHORS OR COPYRIGHT HOLDERS BE LIABLE FOR ANY CLAIM, DAMAGES OR OTHER 
LIABILITY, WHETHER IN AN ACTION OF CONTRACT, TORT OR OTHERWISE, ARISING FROM, 
OUT OF OR IN CONNECTION WITH THE SOFTWARE OR THE USE OR OTHER DEALINGS 
IN THE SOFTWARE.
*)
counter_puls := 0;
puls_temp := 0;
END_ACTION

ACTION SL_SORTING_active:
(*
Copyright (c) 2019 Manuel Goester, Michael Witt, Klaus Kammerer
Institute of Databases and Information Systems, Ulm University, Germany

Permission is hereby granted, free of charge, to any person obtaining a copy 
of this software and associated documentation files (the "Software"), to deal 
in the Software without restriction, including without limitation the rights 
to use, copy, modify, merge, publish, distribute, sublicense, and/or sell 
copies of the Software, and to permit persons to whom the Software is 
furnished to do so, subject to the following conditions:

The above copyright notice and this permission notice shall be included in 
all copies or substantial portions of the Software.

THE SOFTWARE IS PROVIDED "AS IS", WITHOUT WARRANTY OF ANY KIND, EXPRESS OR 
IMPLIED, INCLUDING BUT NOT LIMITED TO THE WARRANTIES OF MERCHANTABILITY, 
FITNESS FOR A PARTICULAR PURPOSE AND NONINFRINGEMENT. IN NO EVENT SHALL THE 
AUTHORS OR COPYRIGHT HOLDERS BE LIABLE FOR ANY CLAIM, DAMAGES OR OTHER 
LIABILITY, WHETHER IN AN ACTION OF CONTRACT, TORT OR OTHERWISE, ARISING FROM, 
OUT OF OR IN CONNECTION WITH THE SOFTWARE OR THE USE OR OTHER DEALINGS 
IN THE SOFTWARE.
*)
SL.mConveyorBelt := TRUE;
IF TC.batchJobQueue.batchJobs[SL.bIdx].workpieces[SL.wIdx].format.colorCheckEnabled THEN
	timer(IN:= TRUE, PT := T#3S);
	IF white AND counter_puls = 35 THEN
		SL.mConveyorBelt := FALSE;
		SL.compressor := TRUE;
		SL.valveFirstEject := TRUE;
	END_IF
	
	IF red AND counter_puls = 45 THEN
		SL.mConveyorBelt := FALSE;
		SL.compressor := TRUE;
		SL.valveSecEject := TRUE;
	END_IF
	
	IF blue AND counter_puls = 55 THEN
		SL.mConveyorBelt := FALSE;
		SL.compressor := TRUE;
		SL.valveThirdEject := TRUE;
	END_IF
	
	IF NOT(timer.Q = FALSE AND timer.IN) THEN
		SL.mConveyorBelt := FALSE;
		SL.compressor := FALSE;	
		SL.valveFirstEject := FALSE;
		SL.valveSecEject := FALSE;
		SL.valveThirdEject := FALSE;
		
		timer(IN:= FALSE);
		
		SL.state := SL_State.SORTING;
	END_IF
ELSE
	timer(IN:= TRUE, PT := T#2S);
	IF counter_puls = 37 THEN
		SL.mConveyorBelt := FALSE;
		SL.compressor := TRUE;
		SL.valveFirstEject := TRUE;
	END_IF
	IF NOT(timer.Q = FALSE AND timer.IN) THEN
		SL.compressor := FALSE;	
		SL.valveFirstEject := FALSE;
		SL.valveSecEject := FALSE;
		SL.valveThirdEject := FALSE;
		
		timer(IN:= FALSE);
		
		SL.state := SL_State.SORTING;
	END_IF
END_IF
END_ACTION

ACTION SL_STOREROOM_active:
(*
Copyright (c) 2019 Manuel Goester, Michael Witt, Klaus Kammerer
Institute of Databases and Information Systems, Ulm University, Germany

Permission is hereby granted, free of charge, to any person obtaining a copy 
of this software and associated documentation files (the "Software"), to deal 
in the Software without restriction, including without limitation the rights 
to use, copy, modify, merge, publish, distribute, sublicense, and/or sell 
copies of the Software, and to permit persons to whom the Software is 
furnished to do so, subject to the following conditions:

The above copyright notice and this permission notice shall be included in 
all copies or substantial portions of the Software.

THE SOFTWARE IS PROVIDED "AS IS", WITHOUT WARRANTY OF ANY KIND, EXPRESS OR 
IMPLIED, INCLUDING BUT NOT LIMITED TO THE WARRANTIES OF MERCHANTABILITY, 
FITNESS FOR A PARTICULAR PURPOSE AND NONINFRINGEMENT. IN NO EVENT SHALL THE 
AUTHORS OR COPYRIGHT HOLDERS BE LIABLE FOR ANY CLAIM, DAMAGES OR OTHER 
LIABILITY, WHETHER IN AN ACTION OF CONTRACT, TORT OR OTHERWISE, ARISING FROM, 
OUT OF OR IN CONNECTION WITH THE SOFTWARE OR THE USE OR OTHER DEALINGS 
IN THE SOFTWARE.
*)
IF white AND NOT(SL.lbWhite) THEN
	rack_white := rack_white + 1;
	SL.state := SL_State.WAITING_FOR_VG_TO_PICK_UP_W;
ELSIF red AND NOT(SL.lbRed) THEN
	rack_red := rack_red + 1;
	SL.state := SL_State.WAITING_FOR_VG_TO_PICK_UP_W;
ELSIF blue AND NOT(SL.lbBlue) THEN
	rack_blue := rack_blue + 1;
	SL.state := SL_State.WAITING_FOR_VG_TO_PICK_UP_W;
ELSE
	// no sorting
	SL.state := SL_State.EJECT;
END_IF
// important! --> signals SL_single/multi_MODE PRG that FB is finished
fin := TRUE;
END_ACTION

END_FUNCTION_BLOCK

// Device/Application/SL/SL_MULTI_MODE
PROGRAM SL_MULTI_MODE
VAR
	fin: BOOL;
	sl_fb: SL_FB;
	step: INT := 1;
END_VAR

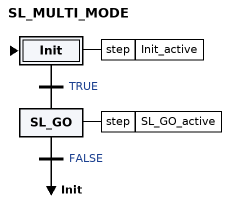
INITIAL_STEP Init:
    Init_active(N);  // step action
END_STEP
TRANSITION FROM Init TO SL_GO
    := TRUE;
END_TRANSITION
STEP SL_GO:
    SL_GO_active(N);  // step action
END_STEP
TRANSITION FROM SL_GO TO Init
    := FALSE;
END_TRANSITION

ACTION SL_GO_active:
(*
Copyright (c) 2019 Manuel Goester, Michael Witt, Klaus Kammerer
Institute of Databases and Information Systems, Ulm University, Germany

Permission is hereby granted, free of charge, to any person obtaining a copy 
of this software and associated documentation files (the "Software"), to deal 
in the Software without restriction, including without limitation the rights 
to use, copy, modify, merge, publish, distribute, sublicense, and/or sell 
copies of the Software, and to permit persons to whom the Software is 
furnished to do so, subject to the following conditions:

The above copyright notice and this permission notice shall be included in 
all copies or substantial portions of the Software.

THE SOFTWARE IS PROVIDED "AS IS", WITHOUT WARRANTY OF ANY KIND, EXPRESS OR 
IMPLIED, INCLUDING BUT NOT LIMITED TO THE WARRANTIES OF MERCHANTABILITY, 
FITNESS FOR A PARTICULAR PURPOSE AND NONINFRINGEMENT. IN NO EVENT SHALL THE 
AUTHORS OR COPYRIGHT HOLDERS BE LIABLE FOR ANY CLAIM, DAMAGES OR OTHER 
LIABILITY, WHETHER IN AN ACTION OF CONTRACT, TORT OR OTHERWISE, ARISING FROM, 
OUT OF OR IN CONNECTION WITH THE SOFTWARE OR THE USE OR OTHER DEALINGS 
IN THE SOFTWARE.
*)
CASE step OF
	1:
		IF SL.currW.state <> W_State.NULL AND SL.state = SL_State.WAITING_FOR_W THEN
			SL.state := SL_State.W_RECEIVED;
			step := step + 1;
		END_IF
	2:
		IF NOT(fin) THEN
			sl_fb();
			fin := sl_fb.fin;
		ELSE
			// wait for VG to pick up w
			SL.state := SL_State.WAITING_FOR_VG_TO_PICK_UP_W;
			step := step + 1;
		END_IF
	3:
		IF VG.state = VG_State.TO_SL_TAKE_W_FINISHED OR SL.state = SL_State.EJECTED THEN
			// finished
			// reset own pointers
			SL.bIdx := 0;
			SL.wIdx := 0;
			SL.currW := TC.nullW;
			// reset fin
			fin := FALSE;
			SL.state := SL_State.WAITING_FOR_W;
			step := 1;
		END_IF
END_CASE
END_ACTION

ACTION Init_active:
(*
Copyright (c) 2019 Manuel Goester, Michael Witt, Klaus Kammerer
Institute of Databases and Information Systems, Ulm University, Germany

Permission is hereby granted, free of charge, to any person obtaining a copy 
of this software and associated documentation files (the "Software"), to deal 
in the Software without restriction, including without limitation the rights 
to use, copy, modify, merge, publish, distribute, sublicense, and/or sell 
copies of the Software, and to permit persons to whom the Software is 
furnished to do so, subject to the following conditions:

The above copyright notice and this permission notice shall be included in 
all copies or substantial portions of the Software.

THE SOFTWARE IS PROVIDED "AS IS", WITHOUT WARRANTY OF ANY KIND, EXPRESS OR 
IMPLIED, INCLUDING BUT NOT LIMITED TO THE WARRANTIES OF MERCHANTABILITY, 
FITNESS FOR A PARTICULAR PURPOSE AND NONINFRINGEMENT. IN NO EVENT SHALL THE 
AUTHORS OR COPYRIGHT HOLDERS BE LIABLE FOR ANY CLAIM, DAMAGES OR OTHER 
LIABILITY, WHETHER IN AN ACTION OF CONTRACT, TORT OR OTHERWISE, ARISING FROM, 
OUT OF OR IN CONNECTION WITH THE SOFTWARE OR THE USE OR OTHER DEALINGS 
IN THE SOFTWARE.
*)
SL.state := SL_State.WAITING_FOR_W;
step := 1;
END_ACTION

END_PROGRAM

// Device/Application/HR/HR_SINGLE_MODE
PROGRAM HR_SINGLE_MODE
VAR
	selectionValid: BOOL;	
	tX: TON;
	tY: TON;
	xFin: BOOL;
	yFin: BOOL;
	zFin: BOOL;
	conveyorBeltFin: BOOL;
	subBlockStart: BOOL;
	fin: BOOL;
	hr_get_w: HR_GET_W;
	hr_store_w: HR_STORE_W;
	hr_put_w_on_conveyor: HR_PUT_W_ON_CONVEYOR;
	
	calibrateYAxis: INT;
	alreadyCounted: BOOL;
	step: INT := 1;
	timer: TON;
END_VAR

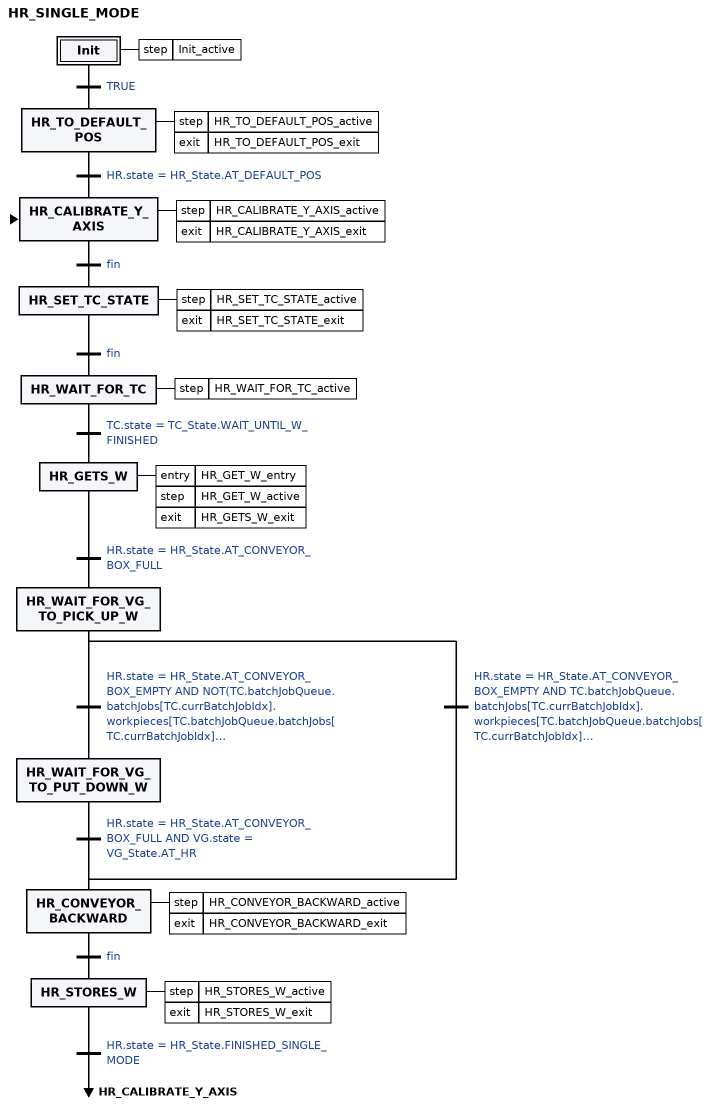
INITIAL_STEP Init:
    Init_active(N);  // step action
END_STEP
TRANSITION FROM Init TO HR_TO_DEFAULT_POS
    := TRUE;
END_TRANSITION
STEP HR_TO_DEFAULT_POS:
    HR_TO_DEFAULT_POS_active(N);  // step action
    HR_TO_DEFAULT_POS_exit(P0);  // exit action
END_STEP
TRANSITION FROM HR_TO_DEFAULT_POS TO HR_CALIBRATE_Y_AXIS
    := HR.state = HR_State.AT_DEFAULT_POS;
END_TRANSITION
STEP HR_CALIBRATE_Y_AXIS:
    HR_CALIBRATE_Y_AXIS_active(N);  // step action
    HR_CALIBRATE_Y_AXIS_exit(P0);  // exit action
END_STEP
TRANSITION FROM HR_CALIBRATE_Y_AXIS TO HR_SET_TC_STATE
    := fin;
END_TRANSITION
STEP HR_SET_TC_STATE:
    HR_SET_TC_STATE_active(N);  // step action
    HR_SET_TC_STATE_exit(P0);  // exit action
END_STEP
TRANSITION FROM HR_SET_TC_STATE TO HR_WAIT_FOR_TC
    := fin;
END_TRANSITION
STEP HR_WAIT_FOR_TC:
    HR_WAIT_FOR_TC_active(N);  // step action
END_STEP
TRANSITION FROM HR_WAIT_FOR_TC TO HR_GETS_W
    := TC.state = TC_State.WAIT_UNTIL_W_FINISHED;
END_TRANSITION
STEP HR_GETS_W:
    HR_GET_W_entry(P1);  // entry action
    HR_GET_W_active(N);  // step action
    HR_GETS_W_exit(P0);  // exit action
END_STEP
TRANSITION FROM HR_GETS_W TO HR_WAIT_FOR_VG_TO_PICK_UP_W
    := HR.state = HR_State.AT_CONVEYOR_BOX_FULL;
END_TRANSITION
STEP HR_WAIT_FOR_VG_TO_PICK_UP_W:
END_STEP
TRANSITION FROM HR_WAIT_FOR_VG_TO_PICK_UP_W TO HR_WAIT_FOR_VG_TO_PUT_DOWN_W
    := HR.state = HR_State.AT_CONVEYOR_BOX_EMPTY AND NOT(TC.batchJobQueue.batchJobs[TC.currBatchJobIdx].workpieces[TC.batchJobQueue.batchJobs[TC.currBatchJobIdx].nextNotProcessedIdx].format.ejectEnabled);
END_TRANSITION
STEP HR_WAIT_FOR_VG_TO_PUT_DOWN_W:
END_STEP
TRANSITION FROM HR_WAIT_FOR_VG_TO_PUT_DOWN_W TO HR_CONVEYOR_BACKWARD
    := HR.state = HR_State.AT_CONVEYOR_BOX_FULL AND VG.state = VG_State.AT_HR;
END_TRANSITION
TRANSITION FROM HR_WAIT_FOR_VG_TO_PICK_UP_W TO HR_CONVEYOR_BACKWARD
    := HR.state = HR_State.AT_CONVEYOR_BOX_EMPTY AND TC.batchJobQueue.batchJobs[TC.currBatchJobIdx].workpieces[TC.batchJobQueue.batchJobs[TC.currBatchJobIdx].nextNotProcessedIdx].format.ejectEnabled;
END_TRANSITION
STEP HR_CONVEYOR_BACKWARD:
    HR_CONVEYOR_BACKWARD_active(N);  // step action
    HR_CONVEYOR_BACKWARD_exit(P0);  // exit action
END_STEP
TRANSITION FROM HR_CONVEYOR_BACKWARD TO HR_STORES_W
    := fin;
END_TRANSITION
STEP HR_STORES_W:
    HR_STORES_W_active(N);  // step action
    HR_STORES_W_exit(P0);  // exit action
END_STEP
TRANSITION FROM HR_STORES_W TO HR_CALIBRATE_Y_AXIS
    := HR.state = HR_State.FINISHED_SINGLE_MODE;
END_TRANSITION

ACTION HR_GET_W_active:
(*
Copyright (c) 2019 Manuel Goester, Michael Witt, Klaus Kammerer
Institute of Databases and Information Systems, Ulm University, Germany

Permission is hereby granted, free of charge, to any person obtaining a copy 
of this software and associated documentation files (the "Software"), to deal 
in the Software without restriction, including without limitation the rights 
to use, copy, modify, merge, publish, distribute, sublicense, and/or sell 
copies of the Software, and to permit persons to whom the Software is 
furnished to do so, subject to the following conditions:

The above copyright notice and this permission notice shall be included in 
all copies or substantial portions of the Software.

THE SOFTWARE IS PROVIDED "AS IS", WITHOUT WARRANTY OF ANY KIND, EXPRESS OR 
IMPLIED, INCLUDING BUT NOT LIMITED TO THE WARRANTIES OF MERCHANTABILITY, 
FITNESS FOR A PARTICULAR PURPOSE AND NONINFRINGEMENT. IN NO EVENT SHALL THE 
AUTHORS OR COPYRIGHT HOLDERS BE LIABLE FOR ANY CLAIM, DAMAGES OR OTHER 
LIABILITY, WHETHER IN AN ACTION OF CONTRACT, TORT OR OTHERWISE, ARISING FROM, 
OUT OF OR IN CONNECTION WITH THE SOFTWARE OR THE USE OR OTHER DEALINGS 
IN THE SOFTWARE.
*)
CASE step OF
	1:
		// get w from rack
		IF NOT fin THEN
			hr_get_w(w:=TC.batchJobQueue.batchJobs[TC.currBatchJobIdx].workpieces[TC.batchJobQueue.batchJobs[TC.currBatchJobIdx].nextNotProcessedIdx]);
			fin := hr_get_w.fin;
		ELSE
			fin := FALSE;
			step := step + 1;
			
		END_IF
	2:
		// put w on conveyor
		hr_put_w_on_conveyor(w := HR.currW);
		fin := hr_put_w_on_conveyor.fin;	
		IF fin THEN
			step := step + 1;
			fin := FALSE;
		END_IF
	3:
		// bring it to VG in conveyor
		IF HR.lbOut THEN
			HR.mCbForward := TRUE;
		ELSE
			// start 1 sec timer to drive conveyor 1 sec longer to be sure that box is at outside pos
			timer(IN:= TRUE, PT := T#1S);
			IF NOT(timer.Q = FALSE AND timer.IN) THEN
				timer(IN:= FALSE);
				HR.mCbForward := FALSE;
				step := step + 1; 
			END_IF
		END_IF
	4:
		// finished
		step := 1;
		HR.state := HR_State.AT_CONVEYOR_BOX_FULL;
END_CASE
END_ACTION

ACTION ConveyorBack_HR_STORE_W_active_exit:
(*
Copyright (c) 2019 Manuel Goester, Michael Witt, Klaus Kammerer
Institute of Databases and Information Systems, Ulm University, Germany

Permission is hereby granted, free of charge, to any person obtaining a copy 
of this software and associated documentation files (the "Software"), to deal 
in the Software without restriction, including without limitation the rights 
to use, copy, modify, merge, publish, distribute, sublicense, and/or sell 
copies of the Software, and to permit persons to whom the Software is 
furnished to do so, subject to the following conditions:

The above copyright notice and this permission notice shall be included in 
all copies or substantial portions of the Software.

THE SOFTWARE IS PROVIDED "AS IS", WITHOUT WARRANTY OF ANY KIND, EXPRESS OR 
IMPLIED, INCLUDING BUT NOT LIMITED TO THE WARRANTIES OF MERCHANTABILITY, 
FITNESS FOR A PARTICULAR PURPOSE AND NONINFRINGEMENT. IN NO EVENT SHALL THE 
AUTHORS OR COPYRIGHT HOLDERS BE LIABLE FOR ANY CLAIM, DAMAGES OR OTHER 
LIABILITY, WHETHER IN AN ACTION OF CONTRACT, TORT OR OTHERWISE, ARISING FROM, 
OUT OF OR IN CONNECTION WITH THE SOFTWARE OR THE USE OR OTHER DEALINGS 
IN THE SOFTWARE.
*)
conveyorBeltFin := FALSE;
END_ACTION

ACTION HR_STORES_W_active:
(*
Copyright (c) 2019 Manuel Goester, Michael Witt, Klaus Kammerer
Institute of Databases and Information Systems, Ulm University, Germany

Permission is hereby granted, free of charge, to any person obtaining a copy 
of this software and associated documentation files (the "Software"), to deal 
in the Software without restriction, including without limitation the rights 
to use, copy, modify, merge, publish, distribute, sublicense, and/or sell 
copies of the Software, and to permit persons to whom the Software is 
furnished to do so, subject to the following conditions:

The above copyright notice and this permission notice shall be included in 
all copies or substantial portions of the Software.

THE SOFTWARE IS PROVIDED "AS IS", WITHOUT WARRANTY OF ANY KIND, EXPRESS OR 
IMPLIED, INCLUDING BUT NOT LIMITED TO THE WARRANTIES OF MERCHANTABILITY, 
FITNESS FOR A PARTICULAR PURPOSE AND NONINFRINGEMENT. IN NO EVENT SHALL THE 
AUTHORS OR COPYRIGHT HOLDERS BE LIABLE FOR ANY CLAIM, DAMAGES OR OTHER 
LIABILITY, WHETHER IN AN ACTION OF CONTRACT, TORT OR OTHERWISE, ARISING FROM, 
OUT OF OR IN CONNECTION WITH THE SOFTWARE OR THE USE OR OTHER DEALINGS 
IN THE SOFTWARE.
*)
IF NOT fin THEN
	HR.state := HR_State.STORE_W;
	hr_store_w(w:=TC.batchJobQueue.batchJobs[TC.currBatchJobIdx].workpieces[TC.batchJobQueue.batchJobs[TC.currBatchJobIdx].nextNotProcessedIdx]);
	fin := hr_store_w.fin;
ELSIF VG.state = VG_State.AT_HR THEN
	// set BatchJobQueue to next workpiece
	HR.state := HR_State.FINISHED_SINGLE_MODE;
	// reset object
	SM.currW := TC.nullW;
	fin := FALSE;
END_IF
END_ACTION

ACTION ConveyorBack_HR_STORE_W_active_active:
(*
Copyright (c) 2019 Manuel Goester, Michael Witt, Klaus Kammerer
Institute of Databases and Information Systems, Ulm University, Germany

Permission is hereby granted, free of charge, to any person obtaining a copy 
of this software and associated documentation files (the "Software"), to deal 
in the Software without restriction, including without limitation the rights 
to use, copy, modify, merge, publish, distribute, sublicense, and/or sell 
copies of the Software, and to permit persons to whom the Software is 
furnished to do so, subject to the following conditions:

The above copyright notice and this permission notice shall be included in 
all copies or substantial portions of the Software.

THE SOFTWARE IS PROVIDED "AS IS", WITHOUT WARRANTY OF ANY KIND, EXPRESS OR 
IMPLIED, INCLUDING BUT NOT LIMITED TO THE WARRANTIES OF MERCHANTABILITY, 
FITNESS FOR A PARTICULAR PURPOSE AND NONINFRINGEMENT. IN NO EVENT SHALL THE 
AUTHORS OR COPYRIGHT HOLDERS BE LIABLE FOR ANY CLAIM, DAMAGES OR OTHER 
LIABILITY, WHETHER IN AN ACTION OF CONTRACT, TORT OR OTHERWISE, ARISING FROM, 
OUT OF OR IN CONNECTION WITH THE SOFTWARE OR THE USE OR OTHER DEALINGS 
IN THE SOFTWARE.
*)
IF HR.lbIn THEN
	HR.mCbBackward := TRUE;
ELSE
	HR.mCbBackward := FALSE;
	conveyorBeltFin := TRUE;
END_IF
END_ACTION

ACTION HR_TO_DEFAULT_POS_active:
(*
Copyright (c) 2019 Manuel Goester, Michael Witt, Klaus Kammerer
Institute of Databases and Information Systems, Ulm University, Germany

Permission is hereby granted, free of charge, to any person obtaining a copy 
of this software and associated documentation files (the "Software"), to deal 
in the Software without restriction, including without limitation the rights 
to use, copy, modify, merge, publish, distribute, sublicense, and/or sell 
copies of the Software, and to permit persons to whom the Software is 
furnished to do so, subject to the following conditions:

The above copyright notice and this permission notice shall be included in 
all copies or substantial portions of the Software.

THE SOFTWARE IS PROVIDED "AS IS", WITHOUT WARRANTY OF ANY KIND, EXPRESS OR 
IMPLIED, INCLUDING BUT NOT LIMITED TO THE WARRANTIES OF MERCHANTABILITY, 
FITNESS FOR A PARTICULAR PURPOSE AND NONINFRINGEMENT. IN NO EVENT SHALL THE 
AUTHORS OR COPYRIGHT HOLDERS BE LIABLE FOR ANY CLAIM, DAMAGES OR OTHER 
LIABILITY, WHETHER IN AN ACTION OF CONTRACT, TORT OR OTHERWISE, ARISING FROM, 
OUT OF OR IN CONNECTION WITH THE SOFTWARE OR THE USE OR OTHER DEALINGS 
IN THE SOFTWARE.
*)

// returns the High Rack TOWER to its default start position
// set "ausleger" arm to default position
IF HR.sCBack = FALSE THEN
	HR.mCBackward := TRUE;
ELSE 
	HR.mCBackward := FALSE;
	// set tower vertical position to max UP as well as horizontal position max RIGHT
	IF HR.sHorizontal = FALSE THEN
		HR.mHorizontalRight := TRUE;
	ELSE
		HR.mHorizontalRight := FALSE;
		HR.cX := 0;
	END_IF
	
	IF HR.sVertical = FALSE THEN
		HR.mVerticalUp := TRUE;
	ELSE
		HR.mVerticalUp := FALSE;
		HR.cY := 0;
	END_IF
END_IF

IF HR.sHorizontal AND HR.sVertical AND HR.sCBack THEN
	HR.state := HR_State.AT_DEFAULT_POS;
END_IF
END_ACTION

ACTION HR_GET_W_entry:
(*
Copyright (c) 2019 Manuel Goester, Michael Witt, Klaus Kammerer
Institute of Databases and Information Systems, Ulm University, Germany

Permission is hereby granted, free of charge, to any person obtaining a copy 
of this software and associated documentation files (the "Software"), to deal 
in the Software without restriction, including without limitation the rights 
to use, copy, modify, merge, publish, distribute, sublicense, and/or sell 
copies of the Software, and to permit persons to whom the Software is 
furnished to do so, subject to the following conditions:

The above copyright notice and this permission notice shall be included in 
all copies or substantial portions of the Software.

THE SOFTWARE IS PROVIDED "AS IS", WITHOUT WARRANTY OF ANY KIND, EXPRESS OR 
IMPLIED, INCLUDING BUT NOT LIMITED TO THE WARRANTIES OF MERCHANTABILITY, 
FITNESS FOR A PARTICULAR PURPOSE AND NONINFRINGEMENT. IN NO EVENT SHALL THE 
AUTHORS OR COPYRIGHT HOLDERS BE LIABLE FOR ANY CLAIM, DAMAGES OR OTHER 
LIABILITY, WHETHER IN AN ACTION OF CONTRACT, TORT OR OTHERWISE, ARISING FROM, 
OUT OF OR IN CONNECTION WITH THE SOFTWARE OR THE USE OR OTHER DEALINGS 
IN THE SOFTWARE.
*)
HR.state := HR_State.GET_W;
END_ACTION

ACTION HR_TO_DEFAULT_POS_exit:
(*
Copyright (c) 2019 Manuel Goester, Michael Witt, Klaus Kammerer
Institute of Databases and Information Systems, Ulm University, Germany

Permission is hereby granted, free of charge, to any person obtaining a copy 
of this software and associated documentation files (the "Software"), to deal 
in the Software without restriction, including without limitation the rights 
to use, copy, modify, merge, publish, distribute, sublicense, and/or sell 
copies of the Software, and to permit persons to whom the Software is 
furnished to do so, subject to the following conditions:

The above copyright notice and this permission notice shall be included in 
all copies or substantial portions of the Software.

THE SOFTWARE IS PROVIDED "AS IS", WITHOUT WARRANTY OF ANY KIND, EXPRESS OR 
IMPLIED, INCLUDING BUT NOT LIMITED TO THE WARRANTIES OF MERCHANTABILITY, 
FITNESS FOR A PARTICULAR PURPOSE AND NONINFRINGEMENT. IN NO EVENT SHALL THE 
AUTHORS OR COPYRIGHT HOLDERS BE LIABLE FOR ANY CLAIM, DAMAGES OR OTHER 
LIABILITY, WHETHER IN AN ACTION OF CONTRACT, TORT OR OTHERWISE, ARISING FROM, 
OUT OF OR IN CONNECTION WITH THE SOFTWARE OR THE USE OR OTHER DEALINGS 
IN THE SOFTWARE.
*)
HR_SINGLE_MODE.subBlockStart := FALSE;
END_ACTION

ACTION HR_GETS_W_exit:
(*
Copyright (c) 2019 Manuel Goester, Michael Witt, Klaus Kammerer
Institute of Databases and Information Systems, Ulm University, Germany

Permission is hereby granted, free of charge, to any person obtaining a copy 
of this software and associated documentation files (the "Software"), to deal 
in the Software without restriction, including without limitation the rights 
to use, copy, modify, merge, publish, distribute, sublicense, and/or sell 
copies of the Software, and to permit persons to whom the Software is 
furnished to do so, subject to the following conditions:

The above copyright notice and this permission notice shall be included in 
all copies or substantial portions of the Software.

THE SOFTWARE IS PROVIDED "AS IS", WITHOUT WARRANTY OF ANY KIND, EXPRESS OR 
IMPLIED, INCLUDING BUT NOT LIMITED TO THE WARRANTIES OF MERCHANTABILITY, 
FITNESS FOR A PARTICULAR PURPOSE AND NONINFRINGEMENT. IN NO EVENT SHALL THE 
AUTHORS OR COPYRIGHT HOLDERS BE LIABLE FOR ANY CLAIM, DAMAGES OR OTHER 
LIABILITY, WHETHER IN AN ACTION OF CONTRACT, TORT OR OTHERWISE, ARISING FROM, 
OUT OF OR IN CONNECTION WITH THE SOFTWARE OR THE USE OR OTHER DEALINGS 
IN THE SOFTWARE.
*)
fin := FALSE;
END_ACTION

ACTION HR_CONVEYOR_BACKWARD_active:
(*
Copyright (c) 2019 Manuel Goester, Michael Witt, Klaus Kammerer
Institute of Databases and Information Systems, Ulm University, Germany

Permission is hereby granted, free of charge, to any person obtaining a copy 
of this software and associated documentation files (the "Software"), to deal 
in the Software without restriction, including without limitation the rights 
to use, copy, modify, merge, publish, distribute, sublicense, and/or sell 
copies of the Software, and to permit persons to whom the Software is 
furnished to do so, subject to the following conditions:

The above copyright notice and this permission notice shall be included in 
all copies or substantial portions of the Software.

THE SOFTWARE IS PROVIDED "AS IS", WITHOUT WARRANTY OF ANY KIND, EXPRESS OR 
IMPLIED, INCLUDING BUT NOT LIMITED TO THE WARRANTIES OF MERCHANTABILITY, 
FITNESS FOR A PARTICULAR PURPOSE AND NONINFRINGEMENT. IN NO EVENT SHALL THE 
AUTHORS OR COPYRIGHT HOLDERS BE LIABLE FOR ANY CLAIM, DAMAGES OR OTHER 
LIABILITY, WHETHER IN AN ACTION OF CONTRACT, TORT OR OTHERWISE, ARISING FROM, 
OUT OF OR IN CONNECTION WITH THE SOFTWARE OR THE USE OR OTHER DEALINGS 
IN THE SOFTWARE.
*)
IF HR.lbIn THEN
	HR.mCbBackward := TRUE;
ELSE
	HR.mCbBackward := FALSE;
	fin := TRUE;
END_IF
END_ACTION

ACTION Store_W_active:
(*
Copyright (c) 2019 Manuel Goester, Michael Witt, Klaus Kammerer
Institute of Databases and Information Systems, Ulm University, Germany

Permission is hereby granted, free of charge, to any person obtaining a copy 
of this software and associated documentation files (the "Software"), to deal 
in the Software without restriction, including without limitation the rights 
to use, copy, modify, merge, publish, distribute, sublicense, and/or sell 
copies of the Software, and to permit persons to whom the Software is 
furnished to do so, subject to the following conditions:

The above copyright notice and this permission notice shall be included in 
all copies or substantial portions of the Software.

THE SOFTWARE IS PROVIDED "AS IS", WITHOUT WARRANTY OF ANY KIND, EXPRESS OR 
IMPLIED, INCLUDING BUT NOT LIMITED TO THE WARRANTIES OF MERCHANTABILITY, 
FITNESS FOR A PARTICULAR PURPOSE AND NONINFRINGEMENT. IN NO EVENT SHALL THE 
AUTHORS OR COPYRIGHT HOLDERS BE LIABLE FOR ANY CLAIM, DAMAGES OR OTHER 
LIABILITY, WHETHER IN AN ACTION OF CONTRACT, TORT OR OTHERWISE, ARISING FROM, 
OUT OF OR IN CONNECTION WITH THE SOFTWARE OR THE USE OR OTHER DEALINGS 
IN THE SOFTWARE.
*)
IF NOT hr_store_w.fin THEN
	hr_store_w(w:=TC.batchJobQueue.batchJobs[TC.currBatchJobIdx].workpieces[TC.batchJobQueue.batchJobs[TC.currBatchJobIdx].nextNotProcessedIdx]);
ELSE
	HR_SINGLE_MODE.subBlockStart := FALSE;
	
	// set BatchJobQueue to next workpiece

	HR.state := HR_State.FINISHED_SINGLE_MODE;
END_IF
END_ACTION

ACTION ToDefaultPos_HR_STORE_W_active_active:
(*
Copyright (c) 2019 Manuel Goester, Michael Witt, Klaus Kammerer
Institute of Databases and Information Systems, Ulm University, Germany

Permission is hereby granted, free of charge, to any person obtaining a copy 
of this software and associated documentation files (the "Software"), to deal 
in the Software without restriction, including without limitation the rights 
to use, copy, modify, merge, publish, distribute, sublicense, and/or sell 
copies of the Software, and to permit persons to whom the Software is 
furnished to do so, subject to the following conditions:

The above copyright notice and this permission notice shall be included in 
all copies or substantial portions of the Software.

THE SOFTWARE IS PROVIDED "AS IS", WITHOUT WARRANTY OF ANY KIND, EXPRESS OR 
IMPLIED, INCLUDING BUT NOT LIMITED TO THE WARRANTIES OF MERCHANTABILITY, 
FITNESS FOR A PARTICULAR PURPOSE AND NONINFRINGEMENT. IN NO EVENT SHALL THE 
AUTHORS OR COPYRIGHT HOLDERS BE LIABLE FOR ANY CLAIM, DAMAGES OR OTHER 
LIABILITY, WHETHER IN AN ACTION OF CONTRACT, TORT OR OTHERWISE, ARISING FROM, 
OUT OF OR IN CONNECTION WITH THE SOFTWARE OR THE USE OR OTHER DEALINGS 
IN THE SOFTWARE.
*)
// returns the high rack TOWER to its default start position
// set "ausleger" arm to default position
IF HR.sCBack = FALSE THEN
	HR.mCBackward := TRUE;
ELSE 
	HR.mCBackward := FALSE;
	// set tower vertical position to max UP as well as horizontal position max RIGHT
	IF HR.sHorizontal = FALSE THEN
		HR.mHorizontalRight := TRUE;
	ELSE
		HR.mHorizontalRight := FALSE;
	END_IF
	
	IF HR.sVertical = FALSE THEN
		HR.mVerticalUp := TRUE;
	ELSE
		HR.mVerticalUp := FALSE;
	END_IF
END_IF
END_ACTION

ACTION HR_WAIT_FOR_TC_active:

END_ACTION

ACTION HR_CONVEYOR_BACKWARD_exit:
(*
Copyright (c) 2019 Manuel Goester, Michael Witt, Klaus Kammerer
Institute of Databases and Information Systems, Ulm University, Germany

Permission is hereby granted, free of charge, to any person obtaining a copy 
of this software and associated documentation files (the "Software"), to deal 
in the Software without restriction, including without limitation the rights 
to use, copy, modify, merge, publish, distribute, sublicense, and/or sell 
copies of the Software, and to permit persons to whom the Software is 
furnished to do so, subject to the following conditions:

The above copyright notice and this permission notice shall be included in 
all copies or substantial portions of the Software.

THE SOFTWARE IS PROVIDED "AS IS", WITHOUT WARRANTY OF ANY KIND, EXPRESS OR 
IMPLIED, INCLUDING BUT NOT LIMITED TO THE WARRANTIES OF MERCHANTABILITY, 
FITNESS FOR A PARTICULAR PURPOSE AND NONINFRINGEMENT. IN NO EVENT SHALL THE 
AUTHORS OR COPYRIGHT HOLDERS BE LIABLE FOR ANY CLAIM, DAMAGES OR OTHER 
LIABILITY, WHETHER IN AN ACTION OF CONTRACT, TORT OR OTHERWISE, ARISING FROM, 
OUT OF OR IN CONNECTION WITH THE SOFTWARE OR THE USE OR OTHER DEALINGS 
IN THE SOFTWARE.
*)
fin := FALSE;
END_ACTION

ACTION Init_active:
(*
Copyright (c) 2019 Manuel Goester, Michael Witt, Klaus Kammerer
Institute of Databases and Information Systems, Ulm University, Germany

Permission is hereby granted, free of charge, to any person obtaining a copy 
of this software and associated documentation files (the "Software"), to deal 
in the Software without restriction, including without limitation the rights 
to use, copy, modify, merge, publish, distribute, sublicense, and/or sell 
copies of the Software, and to permit persons to whom the Software is 
furnished to do so, subject to the following conditions:

The above copyright notice and this permission notice shall be included in 
all copies or substantial portions of the Software.

THE SOFTWARE IS PROVIDED "AS IS", WITHOUT WARRANTY OF ANY KIND, EXPRESS OR 
IMPLIED, INCLUDING BUT NOT LIMITED TO THE WARRANTIES OF MERCHANTABILITY, 
FITNESS FOR A PARTICULAR PURPOSE AND NONINFRINGEMENT. IN NO EVENT SHALL THE 
AUTHORS OR COPYRIGHT HOLDERS BE LIABLE FOR ANY CLAIM, DAMAGES OR OTHER 
LIABILITY, WHETHER IN AN ACTION OF CONTRACT, TORT OR OTHERWISE, ARISING FROM, 
OUT OF OR IN CONNECTION WITH THE SOFTWARE OR THE USE OR OTHER DEALINGS 
IN THE SOFTWARE.
*)
selectionValid := FALSE;
xFin := FALSE;
yFin := FALSE;
zFin := FALSE;
conveyorBeltFin := FALSE;
subBlockStart := FALSE;
calibrateYAxis := 0;
step := 1;
END_ACTION

ACTION ConveyorBack_HR_STORE_W_active_entry:
(*
Copyright (c) 2019 Manuel Goester, Michael Witt, Klaus Kammerer
Institute of Databases and Information Systems, Ulm University, Germany

Permission is hereby granted, free of charge, to any person obtaining a copy 
of this software and associated documentation files (the "Software"), to deal 
in the Software without restriction, including without limitation the rights 
to use, copy, modify, merge, publish, distribute, sublicense, and/or sell 
copies of the Software, and to permit persons to whom the Software is 
furnished to do so, subject to the following conditions:

The above copyright notice and this permission notice shall be included in 
all copies or substantial portions of the Software.

THE SOFTWARE IS PROVIDED "AS IS", WITHOUT WARRANTY OF ANY KIND, EXPRESS OR 
IMPLIED, INCLUDING BUT NOT LIMITED TO THE WARRANTIES OF MERCHANTABILITY, 
FITNESS FOR A PARTICULAR PURPOSE AND NONINFRINGEMENT. IN NO EVENT SHALL THE 
AUTHORS OR COPYRIGHT HOLDERS BE LIABLE FOR ANY CLAIM, DAMAGES OR OTHER 
LIABILITY, WHETHER IN AN ACTION OF CONTRACT, TORT OR OTHERWISE, ARISING FROM, 
OUT OF OR IN CONNECTION WITH THE SOFTWARE OR THE USE OR OTHER DEALINGS 
IN THE SOFTWARE.
*)
SM.currW.linePos := 0;
HR.state := HR_State.STORE_W;
END_ACTION

ACTION HR_CALIBRATE_Y_AXIS_active:
(*
Copyright (c) 2019 Manuel Goester, Michael Witt, Klaus Kammerer
Institute of Databases and Information Systems, Ulm University, Germany

Permission is hereby granted, free of charge, to any person obtaining a copy 
of this software and associated documentation files (the "Software"), to deal 
in the Software without restriction, including without limitation the rights 
to use, copy, modify, merge, publish, distribute, sublicense, and/or sell 
copies of the Software, and to permit persons to whom the Software is 
furnished to do so, subject to the following conditions:

The above copyright notice and this permission notice shall be included in 
all copies or substantial portions of the Software.

THE SOFTWARE IS PROVIDED "AS IS", WITHOUT WARRANTY OF ANY KIND, EXPRESS OR 
IMPLIED, INCLUDING BUT NOT LIMITED TO THE WARRANTIES OF MERCHANTABILITY, 
FITNESS FOR A PARTICULAR PURPOSE AND NONINFRINGEMENT. IN NO EVENT SHALL THE 
AUTHORS OR COPYRIGHT HOLDERS BE LIABLE FOR ANY CLAIM, DAMAGES OR OTHER 
LIABILITY, WHETHER IN AN ACTION OF CONTRACT, TORT OR OTHERWISE, ARISING FROM, 
OUT OF OR IN CONNECTION WITH THE SOFTWARE OR THE USE OR OTHER DEALINGS 
IN THE SOFTWARE.
*)
IF calibrateYAxis = 2 THEN
	IF NOT(HR.sVertical) THEN
		HR.mVerticalUp := TRUE;
	ELSE
		Hr.mVerticalUp := FALSE;
		Hr.cY := 0;
		fin := TRUE;
		calibrateYAxis := 0;
	END_IF
ELSE
	IF NOT(alreadyCounted) THEN
		calibrateYAxis := calibrateYAxis + 1;
		alreadyCounted := TRUE;
	ELSE
		fin := TRUE;
	END_IF
END_IF
END_ACTION

ACTION HR_CALIBRATE_Y_AXIS_exit:
(*
Copyright (c) 2019 Manuel Goester, Michael Witt, Klaus Kammerer
Institute of Databases and Information Systems, Ulm University, Germany

Permission is hereby granted, free of charge, to any person obtaining a copy 
of this software and associated documentation files (the "Software"), to deal 
in the Software without restriction, including without limitation the rights 
to use, copy, modify, merge, publish, distribute, sublicense, and/or sell 
copies of the Software, and to permit persons to whom the Software is 
furnished to do so, subject to the following conditions:

The above copyright notice and this permission notice shall be included in 
all copies or substantial portions of the Software.

THE SOFTWARE IS PROVIDED "AS IS", WITHOUT WARRANTY OF ANY KIND, EXPRESS OR 
IMPLIED, INCLUDING BUT NOT LIMITED TO THE WARRANTIES OF MERCHANTABILITY, 
FITNESS FOR A PARTICULAR PURPOSE AND NONINFRINGEMENT. IN NO EVENT SHALL THE 
AUTHORS OR COPYRIGHT HOLDERS BE LIABLE FOR ANY CLAIM, DAMAGES OR OTHER 
LIABILITY, WHETHER IN AN ACTION OF CONTRACT, TORT OR OTHERWISE, ARISING FROM, 
OUT OF OR IN CONNECTION WITH THE SOFTWARE OR THE USE OR OTHER DEALINGS 
IN THE SOFTWARE.
*)
fin := FALSE;
alreadyCounted := FALSE;
END_ACTION

ACTION HR_CONVEYOR_FORWARD_exit:
(*
Copyright (c) 2019 Manuel Goester, Michael Witt, Klaus Kammerer
Institute of Databases and Information Systems, Ulm University, Germany

Permission is hereby granted, free of charge, to any person obtaining a copy 
of this software and associated documentation files (the "Software"), to deal 
in the Software without restriction, including without limitation the rights 
to use, copy, modify, merge, publish, distribute, sublicense, and/or sell 
copies of the Software, and to permit persons to whom the Software is 
furnished to do so, subject to the following conditions:

The above copyright notice and this permission notice shall be included in 
all copies or substantial portions of the Software.

THE SOFTWARE IS PROVIDED "AS IS", WITHOUT WARRANTY OF ANY KIND, EXPRESS OR 
IMPLIED, INCLUDING BUT NOT LIMITED TO THE WARRANTIES OF MERCHANTABILITY, 
FITNESS FOR A PARTICULAR PURPOSE AND NONINFRINGEMENT. IN NO EVENT SHALL THE 
AUTHORS OR COPYRIGHT HOLDERS BE LIABLE FOR ANY CLAIM, DAMAGES OR OTHER 
LIABILITY, WHETHER IN AN ACTION OF CONTRACT, TORT OR OTHERWISE, ARISING FROM, 
OUT OF OR IN CONNECTION WITH THE SOFTWARE OR THE USE OR OTHER DEALINGS 
IN THE SOFTWARE.
*)
fin := FALSE;
END_ACTION

ACTION HR_CONVEYOR_FORWARD_active:
(*
Copyright (c) 2019 Manuel Goester, Michael Witt, Klaus Kammerer
Institute of Databases and Information Systems, Ulm University, Germany

Permission is hereby granted, free of charge, to any person obtaining a copy 
of this software and associated documentation files (the "Software"), to deal 
in the Software without restriction, including without limitation the rights 
to use, copy, modify, merge, publish, distribute, sublicense, and/or sell 
copies of the Software, and to permit persons to whom the Software is 
furnished to do so, subject to the following conditions:

The above copyright notice and this permission notice shall be included in 
all copies or substantial portions of the Software.

THE SOFTWARE IS PROVIDED "AS IS", WITHOUT WARRANTY OF ANY KIND, EXPRESS OR 
IMPLIED, INCLUDING BUT NOT LIMITED TO THE WARRANTIES OF MERCHANTABILITY, 
FITNESS FOR A PARTICULAR PURPOSE AND NONINFRINGEMENT. IN NO EVENT SHALL THE 
AUTHORS OR COPYRIGHT HOLDERS BE LIABLE FOR ANY CLAIM, DAMAGES OR OTHER 
LIABILITY, WHETHER IN AN ACTION OF CONTRACT, TORT OR OTHERWISE, ARISING FROM, 
OUT OF OR IN CONNECTION WITH THE SOFTWARE OR THE USE OR OTHER DEALINGS 
IN THE SOFTWARE.
*)
IF HR.lbOut THEN
	HR.mCbForward := TRUE;
ELSE
	HR.mCbForward := FALSE;
	fin := TRUE; 
END_IF
END_ACTION

ACTION HR_STORES_W_exit:
(*
Copyright (c) 2019 Manuel Goester, Michael Witt, Klaus Kammerer
Institute of Databases and Information Systems, Ulm University, Germany

Permission is hereby granted, free of charge, to any person obtaining a copy 
of this software and associated documentation files (the "Software"), to deal 
in the Software without restriction, including without limitation the rights 
to use, copy, modify, merge, publish, distribute, sublicense, and/or sell 
copies of the Software, and to permit persons to whom the Software is 
furnished to do so, subject to the following conditions:

The above copyright notice and this permission notice shall be included in 
all copies or substantial portions of the Software.

THE SOFTWARE IS PROVIDED "AS IS", WITHOUT WARRANTY OF ANY KIND, EXPRESS OR 
IMPLIED, INCLUDING BUT NOT LIMITED TO THE WARRANTIES OF MERCHANTABILITY, 
FITNESS FOR A PARTICULAR PURPOSE AND NONINFRINGEMENT. IN NO EVENT SHALL THE 
AUTHORS OR COPYRIGHT HOLDERS BE LIABLE FOR ANY CLAIM, DAMAGES OR OTHER 
LIABILITY, WHETHER IN AN ACTION OF CONTRACT, TORT OR OTHERWISE, ARISING FROM, 
OUT OF OR IN CONNECTION WITH THE SOFTWARE OR THE USE OR OTHER DEALINGS 
IN THE SOFTWARE.
*)
fin := FALSE;
END_ACTION

ACTION HR_SET_TC_STATE_exit:
(*
Copyright (c) 2019 Manuel Goester, Michael Witt, Klaus Kammerer
Institute of Databases and Information Systems, Ulm University, Germany

Permission is hereby granted, free of charge, to any person obtaining a copy 
of this software and associated documentation files (the "Software"), to deal 
in the Software without restriction, including without limitation the rights 
to use, copy, modify, merge, publish, distribute, sublicense, and/or sell 
copies of the Software, and to permit persons to whom the Software is 
furnished to do so, subject to the following conditions:

The above copyright notice and this permission notice shall be included in 
all copies or substantial portions of the Software.

THE SOFTWARE IS PROVIDED "AS IS", WITHOUT WARRANTY OF ANY KIND, EXPRESS OR 
IMPLIED, INCLUDING BUT NOT LIMITED TO THE WARRANTIES OF MERCHANTABILITY, 
FITNESS FOR A PARTICULAR PURPOSE AND NONINFRINGEMENT. IN NO EVENT SHALL THE 
AUTHORS OR COPYRIGHT HOLDERS BE LIABLE FOR ANY CLAIM, DAMAGES OR OTHER 
LIABILITY, WHETHER IN AN ACTION OF CONTRACT, TORT OR OTHERWISE, ARISING FROM, 
OUT OF OR IN CONNECTION WITH THE SOFTWARE OR THE USE OR OTHER DEALINGS 
IN THE SOFTWARE.
*)
fin := FALSE;
END_ACTION

ACTION HR_SET_TC_STATE_active:
(*
Copyright (c) 2019 Manuel Goester, Michael Witt, Klaus Kammerer
Institute of Databases and Information Systems, Ulm University, Germany

Permission is hereby granted, free of charge, to any person obtaining a copy 
of this software and associated documentation files (the "Software"), to deal 
in the Software without restriction, including without limitation the rights 
to use, copy, modify, merge, publish, distribute, sublicense, and/or sell 
copies of the Software, and to permit persons to whom the Software is 
furnished to do so, subject to the following conditions:

The above copyright notice and this permission notice shall be included in 
all copies or substantial portions of the Software.

THE SOFTWARE IS PROVIDED "AS IS", WITHOUT WARRANTY OF ANY KIND, EXPRESS OR 
IMPLIED, INCLUDING BUT NOT LIMITED TO THE WARRANTIES OF MERCHANTABILITY, 
FITNESS FOR A PARTICULAR PURPOSE AND NONINFRINGEMENT. IN NO EVENT SHALL THE 
AUTHORS OR COPYRIGHT HOLDERS BE LIABLE FOR ANY CLAIM, DAMAGES OR OTHER 
LIABILITY, WHETHER IN AN ACTION OF CONTRACT, TORT OR OTHERWISE, ARISING FROM, 
OUT OF OR IN CONNECTION WITH THE SOFTWARE OR THE USE OR OTHER DEALINGS 
IN THE SOFTWARE.
*)
IF NOT(fin) THEN
	IF TC.state = TC_State.W_LOADED THEN
		// workpiece was already loaded by a multi mode batchjob which has been running before this batch job
		// so dont load a now one
		// OR
		// the batch job before was a single mode batch job. So this batch job loaded its workpiece itself
		// now it is loaded, so production can start
		// signalise that production starts
		TC.state := TC_State.WAIT_UNTIL_W_FINISHED;
		fin := TRUE;
	ELSE
		// load a new workpiece
		TC.state := TC_State.LOAD_NEXT_W;
	END_IF
END_IF
END_ACTION

END_PROGRAM

// Device/Application/HR/FBs/HR_GET_W
(*
	HR takes a workpiece out of rack and brings it to conveyor
	
Copyright (c) 2019 Manuel Goester, Michael Witt, Klaus Kammerer
Institute of Databases and Information Systems, Ulm University, Germany

Permission is hereby granted, free of charge, to any person obtaining a copy 
of this software and associated documentation files (the "Software"), to deal 
in the Software without restriction, including without limitation the rights 
to use, copy, modify, merge, publish, distribute, sublicense, and/or sell 
copies of the Software, and to permit persons to whom the Software is 
furnished to do so, subject to the following conditions:

The above copyright notice and this permission notice shall be included in 
all copies or substantial portions of the Software.

THE SOFTWARE IS PROVIDED "AS IS", WITHOUT WARRANTY OF ANY KIND, EXPRESS OR 
IMPLIED, INCLUDING BUT NOT LIMITED TO THE WARRANTIES OF MERCHANTABILITY, 
FITNESS FOR A PARTICULAR PURPOSE AND NONINFRINGEMENT. IN NO EVENT SHALL THE 
AUTHORS OR COPYRIGHT HOLDERS BE LIABLE FOR ANY CLAIM, DAMAGES OR OTHER 
LIABILITY, WHETHER IN AN ACTION OF CONTRACT, TORT OR OTHERWISE, ARISING FROM, 
OUT OF OR IN CONNECTION WITH THE SOFTWARE OR THE USE OR OTHER DEALINGS 
IN THE SOFTWARE.
*)
FUNCTION_BLOCK HR_GET_W
VAR_INPUT
	// the workpiece
	w: Workpiece;
END_VAR
VAR_OUTPUT
END_VAR
VAR
	hr_move: HR_MOVE;
	hr_move_to_pos: HR_MOVE_TO_POS;
	hr_take_w: HR_TAKE_W;
	hr_put_w_on_conveyor: HR_PUT_W_ON_CONVEYOR;
	
	step: INT := 1;
	fin: BOOL := FALSE;
	stepFin: BOOL := FALSE;
END_VAR

CASE step OF
	1: 	// to rack
		fin := FALSE;
		hr_move_to_pos(pos := w.startPos, upOrDown := RackPos.DOWN);
		stepFin := hr_move_to_pos.fin; 
		IF stepFin THEN
			step := step + 1;
			stepFin := FALSE;
		END_IF
	2:	// take w from rack
		hr_take_w(w := w);
		stepFin := hr_take_w.fin;
		IF stepFin THEN
			step := step + 1;
			stepFin := FALSE;
		END_IF
	3:	// to conveyor
		hr_move_to_pos(pos := RackPos.CONVEYOR, upOrDown := RackPos.UP);
		stepFin := hr_move_to_pos.fin;	
		IF stepFin THEN
			step := step + 1;
			stepFin := FALSE;
		END_IF
	
	4:	// finished
		fin := TRUE;
		step := 1;
		stepFin := FALSE;
END_CASE

END_FUNCTION_BLOCK

// Device/Application/HR/FBs/HR_MOVE_TO_POS
(*
	Moves HR to certain position

Copyright (c) 2019 Manuel Goester, Michael Witt, Klaus Kammerer
Institute of Databases and Information Systems, Ulm University, Germany

Permission is hereby granted, free of charge, to any person obtaining a copy 
of this software and associated documentation files (the "Software"), to deal 
in the Software without restriction, including without limitation the rights 
to use, copy, modify, merge, publish, distribute, sublicense, and/or sell 
copies of the Software, and to permit persons to whom the Software is 
furnished to do so, subject to the following conditions:

The above copyright notice and this permission notice shall be included in 
all copies or substantial portions of the Software.

THE SOFTWARE IS PROVIDED "AS IS", WITHOUT WARRANTY OF ANY KIND, EXPRESS OR 
IMPLIED, INCLUDING BUT NOT LIMITED TO THE WARRANTIES OF MERCHANTABILITY, 
FITNESS FOR A PARTICULAR PURPOSE AND NONINFRINGEMENT. IN NO EVENT SHALL THE 
AUTHORS OR COPYRIGHT HOLDERS BE LIABLE FOR ANY CLAIM, DAMAGES OR OTHER 
LIABILITY, WHETHER IN AN ACTION OF CONTRACT, TORT OR OTHERWISE, ARISING FROM, 
OUT OF OR IN CONNECTION WITH THE SOFTWARE OR THE USE OR OTHER DEALINGS 
IN THE SOFTWARE.
*)
FUNCTION_BLOCK HR_MOVE_TO_POS
VAR_INPUT
	// the position where to go
	pos: RackPos;
	// the upper (RackPos.UP) or lower (RackPos.DOWN) position at pos
	upOrDown: RackPos;
END_VAR
VAR_OUTPUT
END_VAR
VAR
	x: INT;
	y: INT;
	// finish flags
	xFin: BOOL := FALSE;
	yFin: BOOL := FALSE;
	fin: BOOL := FALSE;
	// true, if an impulse coming from the motor has been already counted
	xAlreadyCounted: BOOL := FALSE;
	yAlreadyCounted: BOOL := FALSE;
END_VAR

fin := FALSE;

// choose x and y values dependent on the position
CASE pos OF
	RackPos.RACK_11:
		x := 292;
		IF upOrDown = RackPos.DOWN THEN
			y := 17;
		ELSIF upOrDown = RackPos.UP THEN
			y := 1;
		END_IF
	RackPos.RACK_12:
		x := 203;
		IF upOrDown = RackPos.DOWN THEN
			y := 17;
		ELSIF upOrDown = RackPos.UP THEN
			y := 1;
		END_IF
	RackPos.RACK_13:
		x := 114;
		IF upOrDown = RackPos.DOWN THEN
			y := 17;
		ELSIF upOrDown = RackPos.UP THEN
			y := 1;
		END_IF
	RackPos.RACK_21:
		x := 292;
		IF upOrDown = RackPos.DOWN THEN
			y := 70;
		ELSIF upOrDown = RackPos.UP THEN
			y := 54;
		END_IF
	RackPos.RACK_22:
		x := 203;
		IF upOrDown = RackPos.DOWN THEN
			y := 70;
		ELSIF upOrDown = RackPos.UP THEN
			y := 54;
		END_IF
	RackPos.RACK_23:
		x := 114;
		IF upOrDown = RackPos.DOWN THEN
			y := 70;
		ELSIF upOrDown = RackPos.UP THEN
			y := 54;
		END_IF
	RackPos.RACK_31:
		x := 292;
		IF upOrDown = RackPos.DOWN THEN
			y := 129;
		ELSIF upOrDown = RackPos.UP THEN
			y := 113;
		END_IF
	RackPos.RACK_32:
		x := 203;
		IF upOrDown = RackPos.DOWN THEN
			y := 129;
		ELSIF upOrDown = RackPos.UP THEN
			y := 113;
		END_IF
	RackPos.RACK_33:
		x := 114;
		IF upOrDown = RackPos.DOWN THEN
			y := 129;
		ELSIF upOrDown = RackPos.UP THEN
			y := 113;
		END_IF
	RackPos.CONVEYOR:
		x := 0;
		IF upOrDown = RackPos.DOWN THEN
			y := 112;
		ELSIF upOrDown = RackPos.UP THEN
			y := 96;
		END_IF
END_CASE;

// to handle negative counter values
IF HR.cX < 0 THEN
	HR.cX := 0;
END_IF
IF HR.cY < 0 THEN
	HR.cY := 0;
END_IF

// X AXIS
IF HR.cX = x THEN
	// if counter reached demanded position, we're done
	HR.mHorizontalRight := FALSE;
	HR.mHorizontalLeft := FALSE;
	xFin := TRUE;
ELSE
	// SAVETY FIRST: HR does not move in x direction if cantilever is not driven back
	IF NOT(HR.sCBack) THEN
		HR.mCBackward := TRUE;
	ELSE
		HR.mCBackward := FALSE;
		xFin := FALSE;
		IF HR.cX < x AND NOT(xFin) THEN
			HR.mHorizontalLeft := TRUE;
			HR.mHorizontalRight := FALSE;
			IF HR.encHorizontal AND NOT(xAlreadyCounted) THEN
				HR.cX := HR.cX + 1;
				xAlreadyCounted := TRUE;
			ELSIF NOT(HR.encHorizontal) THEN
				xAlreadyCounted := FALSE;
			END_IF
		ELSIF HR.cX > x AND NOT(xFin) THEN
			HR.mHorizontalRight := TRUE;
			HR.mHorizontalLeft := FALSE;
			IF HR.encHorizontal AND NOT(xAlreadyCounted) THEN
				HR.cX := HR.cX - 1;
				xAlreadyCounted := TRUE;
			ELSIF NOT(HR.encHorizontal) THEN
				xAlreadyCounted := FALSE;
			END_IF
		END_IF
	END_IF
END_IF




// Y AXIS
IF HR.cY = y THEN
	// if counter reached demanded position, we're done
	HR.mVerticalUp := FALSE;
	HR.mVerticalDown := FALSE;
	yFin := TRUE;
ELSE
	yFin := FALSE;
	IF HR.cY < y AND NOT(yFin) THEN
		HR.mVerticalDown := TRUE;
		HR.mVerticalUp := FALSE;
		IF HR.encVertical AND NOT(yAlreadyCounted) THEN
			HR.cY := HR.cY + 1;
			yAlreadyCounted := TRUE;
		ELSIF NOT(HR.encVertical) THEN
			yAlreadyCounted := FALSE;
		END_IF
	ELSIF HR.cY > y AND NOT(yFin) THEN
		HR.mVerticalUp := TRUE;
		HR.mVerticalDown := FALSE;
		IF HR.encVertical AND NOT(yAlreadyCounted) THEN
			HR.cY := HR.cY - 1;
			yAlreadyCounted := TRUE;
		ELSIF NOT(HR.encVertical) THEN
			yAlreadyCounted := FALSE;
		END_IF
	END_IF
END_IF

// if x and y axis are finsihed, we're done
IF xFin AND yFin THEN
	xFin := FALSE;
	yFin := FALSE;
	fin := TRUE;
	RETURN;
END_IF

END_FUNCTION_BLOCK

// Device/Application/HR/FBs/HR_TAKE_W
(*
	Picks up a workpiece

Copyright (c) 2019 Manuel Goester, Michael Witt, Klaus Kammerer
Institute of Databases and Information Systems, Ulm University, Germany

Permission is hereby granted, free of charge, to any person obtaining a copy 
of this software and associated documentation files (the "Software"), to deal 
in the Software without restriction, including without limitation the rights 
to use, copy, modify, merge, publish, distribute, sublicense, and/or sell 
copies of the Software, and to permit persons to whom the Software is 
furnished to do so, subject to the following conditions:

The above copyright notice and this permission notice shall be included in 
all copies or substantial portions of the Software.

THE SOFTWARE IS PROVIDED "AS IS", WITHOUT WARRANTY OF ANY KIND, EXPRESS OR 
IMPLIED, INCLUDING BUT NOT LIMITED TO THE WARRANTIES OF MERCHANTABILITY, 
FITNESS FOR A PARTICULAR PURPOSE AND NONINFRINGEMENT. IN NO EVENT SHALL THE 
AUTHORS OR COPYRIGHT HOLDERS BE LIABLE FOR ANY CLAIM, DAMAGES OR OTHER 
LIABILITY, WHETHER IN AN ACTION OF CONTRACT, TORT OR OTHERWISE, ARISING FROM, 
OUT OF OR IN CONNECTION WITH THE SOFTWARE OR THE USE OR OTHER DEALINGS 
IN THE SOFTWARE.
*)
FUNCTION_BLOCK HR_TAKE_W
VAR_INPUT
	// The workpiece
	w: Workpiece;
END_VAR
VAR_OUTPUT
END_VAR
VAR
	step: INT := 1;
	hr_move: HR_MOVE;
	fin: BOOL := FALSE;
	stepFin: BOOL := FALSE;
END_VAR

fin := FALSE;
CASE step OF
	1:	// forward
		IF NOT(HR.sCFront) THEN
			HR.mCForward := TRUE;
		ELSE
			HR.mCForward := FALSE;
			step := step + 1;
		END_IF
	2:	// up
		hr_move(x := 0, y := -16);
		stepFin := hr_move.fin;
		IF stepFin THEN
			step := step + 1;
			stepFin := FALSE;
		END_IF
	3:	// step 3: back
		IF NOT(HR.sCBack) THEN
			HR.mCBackward := TRUE;
		ELSE
			HR.mCBackward := FALSE;
			step := step + 1;
		END_IF
	4:	// finished
		fin := TRUE;
		step := 1;
		stepFin := FALSE;	
END_CASE

END_FUNCTION_BLOCK

// Device/Application/HR/FBs/HR_MOVE
(*
	Moves HR in x and y axis
	
Copyright (c) 2019 Manuel Goester, Michael Witt, Klaus Kammerer
Institute of Databases and Information Systems, Ulm University, Germany

Permission is hereby granted, free of charge, to any person obtaining a copy 
of this software and associated documentation files (the "Software"), to deal 
in the Software without restriction, including without limitation the rights 
to use, copy, modify, merge, publish, distribute, sublicense, and/or sell 
copies of the Software, and to permit persons to whom the Software is 
furnished to do so, subject to the following conditions:

The above copyright notice and this permission notice shall be included in 
all copies or substantial portions of the Software.

THE SOFTWARE IS PROVIDED "AS IS", WITHOUT WARRANTY OF ANY KIND, EXPRESS OR 
IMPLIED, INCLUDING BUT NOT LIMITED TO THE WARRANTIES OF MERCHANTABILITY, 
FITNESS FOR A PARTICULAR PURPOSE AND NONINFRINGEMENT. IN NO EVENT SHALL THE 
AUTHORS OR COPYRIGHT HOLDERS BE LIABLE FOR ANY CLAIM, DAMAGES OR OTHER 
LIABILITY, WHETHER IN AN ACTION OF CONTRACT, TORT OR OTHERWISE, ARISING FROM, 
OUT OF OR IN CONNECTION WITH THE SOFTWARE OR THE USE OR OTHER DEALINGS 
IN THE SOFTWARE.
*)
FUNCTION_BLOCK HR_MOVE
VAR_INPUT
	// distance HR will go right (negative value) or left (positive value)
	x: INT;
	// distance HR will go up (negative value) or down (positive value)
	y: INT;
END_VAR
VAR_OUTPUT
	
END_VAR
VAR	
	// finish flags
	xFin: BOOL := FALSE;
	yFin: BOOL := FALSE;
	fin: BOOL := FALSE;
	// true, if an impulse coming from the motor has been already counted
	xAlreadyCounted: BOOL := FALSE;
	yAlreadyCounted: BOOL := FALSE;
	// counters for x and y axis
	cX: INT := 0;
	cY: INT := 0;
END_VAR

fin := FALSE;

// X AXIS
IF x < 0 THEN
	// drive right
	IF cX = x THEN
		// if counter reached demanded position, we're done
		HR.mHorizontalRight := FALSE;
		HR.mHorizontalLeft := FALSE;
		xFin := TRUE;
	ELSE
		xFin := FALSE;
		IF cX > x THEN
			HR.mHorizontalRight := TRUE;
			IF HR.encHorizontal AND NOT(xAlreadyCounted) THEN
				// update local counter
				cX := cX - 1;
				// update global counter
				HR.cX := HR.cX - 1;
				xAlreadyCounted := TRUE;
			ELSIF NOT(HR.encHorizontal) THEN
				xAlreadyCounted := FALSE;
			END_IF
		END_IF
	END_IF
ELSE
	// x >= 0
	// drive left
	IF cX = x THEN
		// if counter reached demanded position, we're done
		HR.mHorizontalRight := FALSE;
		HR.mHorizontalLeft := FALSE;
		xFin := TRUE;
	ELSE
		xFin := FALSE;
		IF cX < x THEN
			HR.mHorizontalLeft := TRUE;
			IF HR.encHorizontal AND NOT(xAlreadyCounted) THEN
				// update local counter
				cX := cX + 1;
				// update global counter
				HR.cX := HR.cX + 1;
				xAlreadyCounted := TRUE;
			ELSIF NOT(HR.encHorizontal) THEN
				xAlreadyCounted := FALSE;
			END_IF
		END_IF
	END_IF
END_IF

// Y AXIS
IF y < 0 THEN
	// drive up
	IF cY = y THEN
		// if counter reached demanded position, we're done
		HR.mVerticalUp := FALSE;
		HR.mVerticalDown := FALSE;
		yFin := TRUE;
	ELSE
		yFin := FALSE;
		IF cY > y THEN
			HR.mVerticalUp := TRUE;
			IF HR.encVertical AND NOT(yAlreadyCounted) THEN
				// update local counter
				cY := cY - 1;
				// update global counter
				HR.cY := HR.cY - 1;
				yAlreadyCounted := TRUE;
			ELSIF NOT(HR.encVertical) THEN
				yAlreadyCounted := FALSE;
			END_IF
		END_IF
	END_IF
ELSE
	// y >= 0
	// drive down
	IF cY = y THEN
		// if counter reached demanded position, we're done
		HR.mVerticalDown := FALSE;
		HR.mVerticalUp := FALSE;
	yFin := TRUE;
	ELSE
		yFin := FALSE;
		IF cY < y THEN
			HR.mVerticalDown := TRUE;
			IF HR.encVertical AND NOT(yAlreadyCounted) THEN
				// update local counter
				cY := cY + 1;
				// update global counter
				HR.cY := HR.cY + 1;
				yAlreadyCounted := TRUE;
			ELSIF NOT(HR.encVertical) THEN
				yAlreadyCounted := FALSE;
			END_IF
		END_IF
	END_IF
END_IF

// if x and y axis are finsihed, we're done
IF xFin AND yFin THEN
	// reset local counters
	cX := 0;
	cY := 0;
	xFin := FALSE;
	yFin := FALSE;
	fin := TRUE;
	RETURN;
END_IF

END_FUNCTION_BLOCK

// Device/Application/HR/FBs/HR_PUT_W_ON_CONVEYOR
(*
	HR puts down a workpiece at conveyor
	
Copyright (c) 2019 Manuel Goester, Michael Witt, Klaus Kammerer
Institute of Databases and Information Systems, Ulm University, Germany

Permission is hereby granted, free of charge, to any person obtaining a copy 
of this software and associated documentation files (the "Software"), to deal 
in the Software without restriction, including without limitation the rights 
to use, copy, modify, merge, publish, distribute, sublicense, and/or sell 
copies of the Software, and to permit persons to whom the Software is 
furnished to do so, subject to the following conditions:

The above copyright notice and this permission notice shall be included in 
all copies or substantial portions of the Software.

THE SOFTWARE IS PROVIDED "AS IS", WITHOUT WARRANTY OF ANY KIND, EXPRESS OR 
IMPLIED, INCLUDING BUT NOT LIMITED TO THE WARRANTIES OF MERCHANTABILITY, 
FITNESS FOR A PARTICULAR PURPOSE AND NONINFRINGEMENT. IN NO EVENT SHALL THE 
AUTHORS OR COPYRIGHT HOLDERS BE LIABLE FOR ANY CLAIM, DAMAGES OR OTHER 
LIABILITY, WHETHER IN AN ACTION OF CONTRACT, TORT OR OTHERWISE, ARISING FROM, 
OUT OF OR IN CONNECTION WITH THE SOFTWARE OR THE USE OR OTHER DEALINGS 
IN THE SOFTWARE.
*)
FUNCTION_BLOCK HR_PUT_W_ON_CONVEYOR
VAR_INPUT
	// The workpiece
	w: Workpiece;
END_VAR
VAR_OUTPUT
END_VAR
VAR
	step: INT := 1;
	hr_move: HR_MOVE;
	fin: BOOL := FALSE;
	stepFin: BOOL := FALSE;
END_VAR

CASE step OF
	1:	// forward
		fin := FALSE;	
		IF NOT(HR.sCFront) THEN
			HR.mCForward := TRUE;
		ELSE
			HR.mCForward := FALSE;
			step := step + 1;
		END_IF
	2:	// down
		hr_move(x := 0 , y := 26);
		stepFin := hr_move.fin; 
		IF stepFin THEN
			step := step + 1;
			stepFin := FALSE;
		END_IF
	3:	// finished
		fin := TRUE;
		step := 1;
END_CASE

END_FUNCTION_BLOCK

// Device/Application/HR/FBs/HR_STORE_W
(*
	Stores a workpiece in rack
	
Copyright (c) 2019 Manuel Goester, Michael Witt, Klaus Kammerer
Institute of Databases and Information Systems, Ulm University, Germany

Permission is hereby granted, free of charge, to any person obtaining a copy 
of this software and associated documentation files (the "Software"), to deal 
in the Software without restriction, including without limitation the rights 
to use, copy, modify, merge, publish, distribute, sublicense, and/or sell 
copies of the Software, and to permit persons to whom the Software is 
furnished to do so, subject to the following conditions:

The above copyright notice and this permission notice shall be included in 
all copies or substantial portions of the Software.

THE SOFTWARE IS PROVIDED "AS IS", WITHOUT WARRANTY OF ANY KIND, EXPRESS OR 
IMPLIED, INCLUDING BUT NOT LIMITED TO THE WARRANTIES OF MERCHANTABILITY, 
FITNESS FOR A PARTICULAR PURPOSE AND NONINFRINGEMENT. IN NO EVENT SHALL THE 
AUTHORS OR COPYRIGHT HOLDERS BE LIABLE FOR ANY CLAIM, DAMAGES OR OTHER 
LIABILITY, WHETHER IN AN ACTION OF CONTRACT, TORT OR OTHERWISE, ARISING FROM, 
OUT OF OR IN CONNECTION WITH THE SOFTWARE OR THE USE OR OTHER DEALINGS 
IN THE SOFTWARE.
*)
FUNCTION_BLOCK HR_STORE_W
VAR_INPUT
	w: Workpiece;
END_VAR
VAR_OUTPUT
END_VAR
VAR
	hr_move: HR_MOVE;
	hr_move_to_pos: HR_MOVE_TO_POS;
	hr_take_w_from_conveyor: HR_TAKE_W_FROM_CONVEYOR;
	hr_put_w: HR_PUT_W;
	
	step: INT := 1;
	fin: BOOL;
	stepFin: BOOL := FALSE;
END_VAR

CASE step OF
	1:	// to conveyor if not already there
		fin := FALSE;
		hr_move_to_pos(pos := RackPos.CONVEYOR, upOrDown := RackPos.DOWN);
		stepFin := hr_move_to_pos.fin;
		IF stepFin THEN
			step := step + 1;
			stepFin := FALSE;
		END_IF
	2:	// take w from conveyor
		hr_take_w_from_conveyor(w := w);
		stepFin := hr_take_w_from_conveyor.fin;
		IF stepFin THEN
			step := step + 1;
			stepFin := FALSE;
		END_IF
	3:	// to rack
		hr_move_to_pos(pos := w.endPos, upOrDown := RackPos.UP);
		stepFin := hr_move_to_pos.fin;
		IF stepFin THEN
			step := step + 1;
			stepFin := FALSE;
		END_IF
	4:	// put w into rack
		hr_put_w();
		stepFin := hr_put_w.fin;
		IF stepFin THEN
			step := step + 1;
			stepFin := FALSE;
		END_IF
	5:	// finished
		fin := TRUE;
		step := 1;
END_CASE

END_FUNCTION_BLOCK

// Device/Application/HR/FBs/HR_TAKE_W_FROM_CONVEYOR
(*
	Picks up a workpiece from conveyor
	
